LIN {X 0,Y 417.431,Z 307.432,A -85,B 0,C 180,E1 -10178.471,E2 -10178.471} C_VEL
LIN {X 0,Y 417.765,Z 300.419,A -85,B 0,C 180,E1 -10179.929,E2 -10179.929} C_VEL
LIN {X 0,Y 418.265,Z 291.62,A -85,B 0,C 180,E1 -10181.387,E2 -10181.387} C_VEL
LIN {X 0,Y 418.822,Z 282.602,A -85,B 0,C 180,E1 -10182.6,E2 -10182.6} C_VEL
LIN {X 0,Y 419.415,Z 273.392,A -85,B 0,C 180,E1 -10183.617,E2 -10183.617} C_VEL
LIN {X 0,Y 420.017,Z 263.241,A -85,B 0,C 180,E1 -10184.536,E2 -10184.536} C_VEL
LIN {X 0,Y 420.775,Z 251.442,A -85,B 0,C 180,E1 -10185.376,E2 -10185.376} C_VEL
LIN {X 0,Y 421.386,Z 239.15,A -85,B 0,C 180,E1 -10186.035,E2 -10186.035} C_VEL
LIN {X 0,Y 421.966,Z 225.694,A -85,B 0,C 180,E1 -10186.541,E2 -10186.541} C_VEL
LIN {X 0,Y 422.2,Z 212.111,A -85,B 0,C 180,E1 -10186.843,E2 -10186.843} C_VEL
LIN {X 0,Y 422.884,Z 138.438,A -85,B 0,C 180,E1 -10188.089,E2 -10188.089} C_VEL
LIN {X 0,Y 419.21,Z 111.774,A -85,B 0,C 180,E1 -10188.701,E2 -10188.701} C_VEL
LIN {X 0,Y 420.191,Z 93.552,A -85,B 0,C 180,E1 -10192.106,E2 -10192.106} C_VEL
LIN {X 0,Y 421.025,Z 79.98,A -85,B 0,C 180,E1 -10194.665,E2 -10194.665} C_VEL
LIN {X 0,Y 418.784,Z 67.568,A -85,B 0,C 180,E1 -10197.197,E2 -10197.197} C_VEL
LIN {X 0,Y 418.347,Z 65.37,A -85,B 0,C 180,E1 -10197.691,E2 -10197.691} C_VEL
LIN {X 0,Y 418.212,Z 65.388,A -85,B 0,C 180,E1 -10201.396,E2 -10201.396} C_VEL
LIN {X 0,Y 418.266,Z 65.381,A -85,B 0,C 180,E1 -10204.58,E2 -10204.58} C_VEL
LIN {X 0,Y 418.235,Z 65.39,A -85,B 0,C 180,E1 -10207.834,E2 -10207.834} C_VEL
LIN {X 0,Y 418.223,Z 65.386,A -85,B 0,C 180,E1 -10210.948,E2 -10210.948} C_VEL
LIN {X 0,Y 418.21,Z 65.392,A -85,B 0,C 180,E1 -10213.729,E2 -10213.729} C_VEL
LIN {X 0,Y 418.208,Z 65.387,A -85,B 0,C 180,E1 -10216.448,E2 -10216.448} C_VEL
LIN {X 0,Y 418.222,Z 65.39,A -85,B 0,C 180,E1 -10219.13,E2 -10219.13} C_VEL
LIN {X 0,Y 418.226,Z 65.385,A -85,B 0,C 180,E1 -10222.167,E2 -10222.167} C_VEL
LIN {X 0,Y 418.265,Z 65.385,A -85,B 0,C 180,E1 -10225.42,E2 -10225.42} C_VEL
LIN {X 0,Y 418.211,Z 65.389,A -85,B 0,C 180,E1 -10228.604,E2 -10228.604} C_VEL
LIN {X 0,Y 418.291,Z 65.377,A -85,B 0,C 180,E1 -10231.937,E2 -10231.937} C_VEL
LIN {X 0,Y 418.289,Z 65.381,A -85,B 0,C 180,E1 -10235.163,E2 -10235.163} C_VEL
LIN {X 0,Y 418.233,Z 65.386,A -85,B 0,C 180,E1 -10238.304,E2 -10238.304} C_VEL
LIN {X 0,Y 418.275,Z 65.38,A -85,B 0,C 180,E1 -10241.383,E2 -10241.383} C_VEL
LIN {X 0,Y 418.301,Z 65.381,A -85,B 0,C 180,E1 -10244.406,E2 -10244.406} C_VEL
LIN {X 0,Y 418.355,Z 65.369,A -85,B 0,C 180,E1 -10247.386,E2 -10247.386} C_VEL
LIN {X 0,Y 418.399,Z 65.363,A -85,B 0,C 180,E1 -10251.305,E2 -10251.305} C_VEL
LIN {X 0,Y 418.509,Z 65.356,A -85,B 0,C 180,E1 -10254.217,E2 -10254.217} C_VEL
LIN {X 0,Y 418.539,Z 65.352,A -85,B 0,C 180,E1 -10258.076,E2 -10258.076} C_VEL
LIN {X 0,Y 418.668,Z 65.336,A -85,B 0,C 180,E1 -10260,E2 -10260} C_VEL
LIN {X 0,Y 418.494,Z 65.352,A -85,B 0,C 180,E1 -10262.888,E2 -10262.888} C_VEL
LIN {X 0,Y 418.457,Z 65.356,A -85,B 0,C 180,E1 -10266.516,E2 -10266.516} C_VEL
LIN {X 0,Y 418.338,Z 65.377,A -85,B 0,C 180,E1 -10269.672,E2 -10269.672} C_VEL
LIN {X 0,Y 418.346,Z 65.371,A -85,B 0,C 180,E1 -10273.001,E2 -10273.001} C_VEL
LIN {X 0,Y 418.312,Z 65.374,A -85,B 0,C 180,E1 -10276.735,E2 -10276.735} C_VEL
LIN {X 0,Y 418.27,Z 65.383,A -85,B 0,C 180,E1 -10279.79,E2 -10279.79} C_VEL
LIN {X 0,Y 418.237,Z 65.385,A -85,B 0,C 180,E1 -10282.737,E2 -10282.737} C_VEL
LIN {X 0,Y 418.261,Z 65.382,A -85,B 0,C 180,E1 -10285.905,E2 -10285.905} C_VEL
LIN {X 0,Y 418.269,Z 65.386,A -85,B 0,C 180,E1 -10289.105,E2 -10289.105} C_VEL
LIN {X 0,Y 418.258,Z 65.386,A -85,B 0,C 180,E1 -10292.844,E2 -10292.844} C_VEL
LIN {X 0,Y 418.245,Z 65.383,A -85,B 0,C 180,E1 -10296.238,E2 -10296.238} C_VEL
LIN {X 0,Y 418.21,Z 65.387,A -85,B 0,C 180,E1 -10299.687,E2 -10299.687} C_VEL
LIN {X 0,Y 418.213,Z 65.389,A -85,B 0,C 180,E1 -10302.319,E2 -10302.319} C_VEL
LIN {X 0,Y 418.237,Z 65.386,A -85,B 0,C 180,E1 -10305.109,E2 -10305.109} C_VEL
LIN {X 0,Y 418.236,Z 65.384,A -85,B 0,C 180,E1 -10307.767,E2 -10307.767} C_VEL
LIN {X 0,Y 418.24,Z 65.383,A -85,B 0,C 180,E1 -10311.557,E2 -10311.557} C_VEL
LIN {X 0,Y 418.261,Z 65.381,A -85,B 0,C 180,E1 -10315.159,E2 -10315.159} C_VEL
LIN {X 0,Y 418.248,Z 65.383,A -85,B 0,C 180,E1 -10317.472,E2 -10317.472} C_VEL
LIN {X 0,Y 418.267,Z 65.38,A -85,B 0,C 180,E1 -10320.897,E2 -10320.897} C_VEL
LIN {X 0,Y 418.234,Z 65.391,A -85,B 0,C 180,E1 -10324.094,E2 -10324.094} C_VEL
LIN {X 0,Y 418.233,Z 65.385,A -85,B 0,C 180,E1 -10327.264,E2 -10327.264} C_VEL
LIN {X 0,Y 418.287,Z 65.379,A -85,B 0,C 180,E1 -10330.365,E2 -10330.365} C_VEL
LIN {X 0,Y 418.32,Z 65.376,A -85,B 0,C 180,E1 -10333.405,E2 -10333.405} C_VEL
LIN {X 0,Y 418.343,Z 65.434,A -85,B 0,C 180,E1 -10335.653,E2 -10335.653} C_VEL
LIN {X 0,Y 419.814,Z 74.736,A -85,B 0,C 180,E1 -10337.921,E2 -10337.921} C_VEL
LIN {X 0,Y 419.849,Z 76.846,A -85,B 0,C 180,E1 -10338.412,E2 -10338.412} C_VEL
LIN {X 0,Y 423.359,Z 95.58,A -85,B 0,C 180,E1 -10338.881,E2 -10338.881} C_VEL
LIN {X 0,Y 422.292,Z 183.825,A -85,B 0,C 180,E1 -10340.392,E2 -10340.392} C_VEL
LIN {X 0,Y 422.034,Z 197.591,A -85,B 0,C 180,E1 -10340.837,E2 -10340.837} C_VEL
LIN {X 0,Y 421.56,Z 210.007,A -85,B 0,C 180,E1 -10341.431,E2 -10341.431} C_VEL
LIN {X 0,Y 421.142,Z 221.833,A -85,B 0,C 180,E1 -10342.208,E2 -10342.208} C_VEL
LIN {X 0,Y 420.759,Z 228.414,A -85,B 0,C 180,E1 -10342.732,E2 -10342.732} C_VEL
LIN {X 0,Y 419.76,Z 233.376,A -85,B 0,C 180,E1 -10343.151,E2 -10343.151} C_VEL
LIN {X 0,Y 416.395,Z 241.174,A -85,B 0,C 180,E1 -10343.859,E2 -10343.859} C_VEL
LIN {X 0,Y 413.103,Z 248.473,A -85,B 0,C 180,E1 -10344.664,E2 -10344.664} C_VEL
LIN {X 0,Y 412.224,Z 252.648,A -85,B 0,C 180,E1 -10345.229,E2 -10345.229} C_VEL
LIN {X 0,Y 411.575,Z 261.003,A -85,B 0,C 180,E1 -10346.574,E2 -10346.574} C_VEL
LIN {X 0,Y 411.024,Z 268.36,A -85,B 0,C 180,E1 -10348.041,E2 -10348.041} C_VEL
LIN {X 0,Y 410.67,Z 274.265,A -85,B 0,C 180,E1 -10349.51,E2 -10349.51} C_VEL
LIN {X 0,Y 410.324,Z 278.946,A -85,B 0,C 180,E1 -10350.982,E2 -10350.982} C_VEL
LIN {X 0,Y 410.218,Z 282.523,A -85,B 0,C 180,E1 -10352.455,E2 -10352.455} C_VEL
LIN {X 0,Y 410.051,Z 285.111,A -85,B 0,C 180,E1 -10353.931,E2 -10353.931} C_VEL
LIN {X 0,Y 410.061,Z 286.328,A -85,B 0,C 180,E1 -10354.916,E2 -10354.916} C_VEL
LIN {X 0,Y 410.118,Z 287.328,A -85,B 0,C 180,E1 -10356.318,E2 -10356.318} C_VEL
LIN {X 0,Y 409.997,Z 287.526,A -85,B 0,C 180,E1 -10357.882,E2 -10357.882} C_VEL
LIN {X 0,Y 410.023,Z 287.151,A -85,B 0,C 180,E1 -10358.874,E2 -10358.874} C_VEL
LIN {X 0,Y 410.015,Z 286.357,A -85,B 0,C 180,E1 -10359.87,E2 -10359.87} C_VEL
LIN {X 0,Y 410.13,Z 285.135,A -85,B 0,C 180,E1 -10360.865,E2 -10360.865} C_VEL
LIN {X 0,Y 410.448,Z 282.065,A -85,B 0,C 180,E1 -10362.576,E2 -10362.576} C_VEL
LIN {X 0,Y 410.797,Z 277.448,A -85,B 0,C 180,E1 -10364.364,E2 -10364.364} C_VEL
LIN {X 0,Y 411.381,Z 271.232,A -85,B 0,C 180,E1 -10366.118,E2 -10366.118} C_VEL
LIN {X 0,Y 411.974,Z 264.461,A -85,B 0,C 180,E1 -10367.619,E2 -10367.619} C_VEL
LIN {X 0,Y 412.633,Z 257.443,A -85,B 0,C 180,E1 -10368.882,E2 -10368.882} C_VEL
LIN {X 0,Y 413.43,Z 248.997,A -85,B 0,C 180,E1 -10370.135,E2 -10370.135} C_VEL
LIN {X 0,Y 414.152,Z 239.692,A -85,B 0,C 180,E1 -10371.268,E2 -10371.268} C_VEL
LIN {X 0,Y 414.956,Z 229.493,A -85,B 0,C 180,E1 -10372.27,E2 -10372.27} C_VEL
LIN {X 0,Y 415.733,Z 218.335,A -85,B 0,C 180,E1 -10373.144,E2 -10373.144} C_VEL
LIN {X 0,Y 416.464,Z 205.903,A -85,B 0,C 180,E1 -10373.892,E2 -10373.892} C_VEL
LIN {X 0,Y 416.995,Z 192.882,A -85,B 0,C 180,E1 -10374.445,E2 -10374.445} C_VEL
LIN {X 0,Y 417.333,Z 179.624,A -85,B 0,C 180,E1 -10374.8,E2 -10374.8} C_VEL
LIN {X 0,Y 418.439,Z 96.881,A -85,B 0,C 180,E1 -10376.241,E2 -10376.241} C_VEL
LIN {X 0,Y 414.203,Z 79.905,A -85,B 0,C 180,E1 -10376.788,E2 -10376.788} C_VEL
LIN {X 0,Y 413.433,Z 77.348,A -85,B 0,C 180,E1 -10376.906,E2 -10376.906} C_VEL
LIN {X 0,Y 411.219,Z 66.264,A -85,B 0,C 180,E1 -10379.817,E2 -10379.817} C_VEL
LIN {X 0,Y 411.206,Z 66.265,A -85,B 0,C 180,E1 -10383.156,E2 -10383.156} C_VEL
LIN {X 0,Y 411.191,Z 66.265,A -85,B 0,C 180,E1 -10386.551,E2 -10386.551} C_VEL
LIN {X 0,Y 411.17,Z 66.27,A -85,B 0,C 180,E1 -10389.72,E2 -10389.72} C_VEL
LIN {X 0,Y 411.164,Z 66.268,A -85,B 0,C 180,E1 -10393.135,E2 -10393.135} C_VEL
LIN {X 0,Y 411.166,Z 66.264,A -85,B 0,C 180,E1 -10395.882,E2 -10395.882} C_VEL
LIN {X 0,Y 411.149,Z 66.265,A -85,B 0,C 180,E1 -10398.775,E2 -10398.775} C_VEL
LIN {X 0,Y 411.179,Z 66.266,A -85,B 0,C 180,E1 -10402.024,E2 -10402.024} C_VEL
LIN {X 0,Y 411.202,Z 66.261,A -85,B 0,C 180,E1 -10405.124,E2 -10405.124} C_VEL
LIN {X 0,Y 411.156,Z 66.263,A -85,B 0,C 180,E1 -10408.001,E2 -10408.001} C_VEL
LIN {X 0,Y 411.17,Z 66.266,A -85,B 0,C 180,E1 -10411.406,E2 -10411.406} C_VEL
LIN {X 0,Y 411.19,Z 66.267,A -85,B 0,C 180,E1 -10414.941,E2 -10414.941} C_VEL
LIN {X 0,Y 411.206,Z 66.256,A -85,B 0,C 180,E1 -10417.913,E2 -10417.913} C_VEL
LIN {X 0,Y 411.222,Z 66.258,A -85,B 0,C 180,E1 -10421.051,E2 -10421.051} C_VEL
LIN {X 0,Y 411.25,Z 66.254,A -85,B 0,C 180,E1 -10424.131,E2 -10424.131} C_VEL
LIN {X 0,Y 411.307,Z 66.242,A -85,B 0,C 180,E1 -10427.165,E2 -10427.165} C_VEL
LIN {X 0,Y 411.29,Z 66.251,A -85,B 0,C 180,E1 -10430.161,E2 -10430.161} C_VEL
LIN {X 0,Y 411.389,Z 66.231,A -85,B 0,C 180,E1 -10433.132,E2 -10433.132} C_VEL
LIN {X 0,Y 411.291,Z 66.248,A -85,B 0,C 180,E1 -10435.099,E2 -10435.099} C_VEL
LIN {X 0,Y 411.509,Z 66.227,A -85,B 0,C 180,E1 -10438.042,E2 -10438.042} C_VEL
LIN {X 0,Y 411.439,Z 66.228,A -85,B 0,C 180,E1 -10440.979,E2 -10440.979} C_VEL
LIN {X 0,Y 411.432,Z 66.233,A -85,B 0,C 180,E1 -10442.937,E2 -10442.937} C_VEL
LIN {X 0,Y 411.432,Z 66.227,A -85,B 0,C 180,E1 -10445.882,E2 -10445.882} C_VEL
LIN {X 0,Y 411.32,Z 66.246,A -85,B 0,C 180,E1 -10448.846,E2 -10448.846} C_VEL
LIN {X 0,Y 411.286,Z 66.246,A -85,B 0,C 180,E1 -10451.833,E2 -10451.833} C_VEL
LIN {X 0,Y 411.258,Z 66.253,A -85,B 0,C 180,E1 -10454.853,E2 -10454.853} C_VEL
LIN {X 0,Y 411.246,Z 66.255,A -85,B 0,C 180,E1 -10457.915,E2 -10457.915} C_VEL
LIN {X 0,Y 411.199,Z 66.263,A -85,B 0,C 180,E1 -10461.034,E2 -10461.034} C_VEL
LIN {X 0,Y 411.22,Z 66.259,A -85,B 0,C 180,E1 -10464.216,E2 -10464.216} C_VEL
LIN {X 0,Y 411.261,Z 66.255,A -85,B 0,C 180,E1 -10467.477,E2 -10467.477} C_VEL
LIN {X 0,Y 411.192,Z 66.263,A -85,B 0,C 180,E1 -10470.847,E2 -10470.847} C_VEL
LIN {X 0,Y 411.209,Z 66.26,A -85,B 0,C 180,E1 -10474.333,E2 -10474.333} C_VEL
LIN {X 0,Y 411.195,Z 66.256,A -85,B 0,C 180,E1 -10477.974,E2 -10477.974} C_VEL
LIN {X 0,Y 411.166,Z 66.267,A -85,B 0,C 180,E1 -10481.228,E2 -10481.228} C_VEL
LIN {X 0,Y 411.178,Z 66.268,A -85,B 0,C 180,E1 -10484.49,E2 -10484.49} C_VEL
LIN {X 0,Y 411.18,Z 66.265,A -85,B 0,C 180,E1 -10488.194,E2 -10488.194} C_VEL
LIN {X 0,Y 411.225,Z 66.26,A -85,B 0,C 180,E1 -10490.776,E2 -10490.776} C_VEL
LIN {X 0,Y 411.2,Z 66.259,A -85,B 0,C 180,E1 -10494.471,E2 -10494.471} C_VEL
LIN {X 0,Y 411.21,Z 66.267,A -85,B 0,C 180,E1 -10496.873,E2 -10496.873} C_VEL
LIN {X 0,Y 411.235,Z 66.265,A -85,B 0,C 180,E1 -10500.644,E2 -10500.644} C_VEL
LIN {X 0,Y 411.251,Z 66.323,A -85,B 0,C 180,E1 -10500.882,E2 -10500.882} C_VEL
LIN {X 0,Y 413.861,Z 78.061,A -85,B 0,C 180,E1 -10503.527,E2 -10503.527} C_VEL
LIN {X 0,Y 415.004,Z 84.662,A -85,B 0,C 180,E1 -10504.952,E2 -10504.952} C_VEL
LIN {X 0,Y 413.661,Z 101.777,A -85,B 0,C 180,E1 -10508.313,E2 -10508.313} C_VEL
LIN {X 0,Y 413.058,Z 111.347,A -85,B 0,C 180,E1 -10510.146,E2 -10510.146} C_VEL
LIN {X 0,Y 417.432,Z 136.961,A -85,B 0,C 180,E1 -10510.852,E2 -10510.852} C_VEL
LIN {X 0,Y 417.89,Z 142.841,A -85,B 0,C 180,E1 -10510.983,E2 -10510.983} C_VEL
LIN {X 0,Y 416.919,Z 219.576,A -85,B 0,C 180,E1 -10512.336,E2 -10512.336} C_VEL
LIN {X 0,Y 416.286,Z 232.903,A -85,B 0,C 180,E1 -10512.752,E2 -10512.752} C_VEL
LIN {X 0,Y 415.492,Z 245.646,A -85,B 0,C 180,E1 -10513.351,E2 -10513.351} C_VEL
LIN {X 0,Y 414.638,Z 257.78,A -85,B 0,C 180,E1 -10514.138,E2 -10514.138} C_VEL
LIN {X 0,Y 413.688,Z 269.312,A -85,B 0,C 180,E1 -10515.11,E2 -10515.11} C_VEL
LIN {X 0,Y 412.753,Z 279.713,A -85,B 0,C 180,E1 -10516.209,E2 -10516.209} C_VEL
LIN {X 0,Y 412.052,Z 289.098,A -85,B 0,C 180,E1 -10517.439,E2 -10517.439} C_VEL
LIN {X 0,Y 411.212,Z 298.174,A -85,B 0,C 180,E1 -10518.914,E2 -10518.914} C_VEL
LIN {X 0,Y 410.659,Z 305.511,A -85,B 0,C 180,E1 -10520.394,E2 -10520.394} C_VEL
LIN {X 0,Y 410.257,Z 312.261,A -85,B 0,C 180,E1 -10522.123,E2 -10522.123} C_VEL
LIN {X 0,Y 410.047,Z 317.157,A -85,B 0,C 180,E1 -10523.77,E2 -10523.77} C_VEL
LIN {X 0,Y 410.002,Z 320.138,A -85,B 0,C 180,E1 -10525.083,E2 -10525.083} C_VEL
LIN {X 0,Y 409.97,Z 323.132,A -85,B 0,C 180,E1 -10527.052,E2 -10527.052} C_VEL
LIN {X 0,Y 410.02,Z 324.037,A -85,B 0,C 180,E1 -10528.035,E2 -10528.035} C_VEL
LIN {X 0,Y 409.984,Z 324.507,A -85,B 0,C 180,E1 -10529.017,E2 -10529.017} C_VEL
LIN {X 0,Y 409.981,Z 324.574,A -85,B 0,C 180,E1 -10530,E2 -10530} C_VEL
LIN {X 0,Y 410.024,Z 323.546,A -85,B 0,C 180,E1 -10531.964,E2 -10531.964} C_VEL
LIN {X 0,Y 410.012,Z 322.408,A -85,B 0,C 180,E1 -10532.947,E2 -10532.947} C_VEL
LIN {X 0,Y 409.959,Z 320.83,A -85,B 0,C 180,E1 -10533.932,E2 -10533.932} C_VEL
LIN {X 0,Y 410,Z 317.661,A -85,B 0,C 180,E1 -10535.409,E2 -10535.409} C_VEL
LIN {X 0,Y 410.076,Z 313.415,A -85,B 0,C 180,E1 -10536.89,E2 -10536.89} C_VEL
LIN {X 0,Y 410.353,Z 306.957,A -85,B 0,C 180,E1 -10538.618,E2 -10538.618} C_VEL
LIN {X 0,Y 410.702,Z 299.897,A -85,B 0,C 180,E1 -10540.102,E2 -10540.102} C_VEL
LIN {X 0,Y 411.266,Z 291.048,A -85,B 0,C 180,E1 -10541.583,E2 -10541.583} C_VEL
LIN {X 0,Y 411.876,Z 281.981,A -85,B 0,C 180,E1 -10542.816,E2 -10542.816} C_VEL
LIN {X 0,Y 412.549,Z 272.003,A -85,B 0,C 180,E1 -10543.923,E2 -10543.923} C_VEL
LIN {X 0,Y 413.228,Z 260.922,A -85,B 0,C 180,E1 -10544.906,E2 -10544.906} C_VEL
LIN {X 0,Y 413.978,Z 248.494,A -85,B 0,C 180,E1 -10545.761,E2 -10545.761} C_VEL
LIN {X 0,Y 414.567,Z 236.704,A -85,B 0,C 180,E1 -10546.37,E2 -10546.37} C_VEL
LIN {X 0,Y 415.167,Z 224.022,A -85,B 0,C 180,E1 -10546.82,E2 -10546.82} C_VEL
LIN {X 0,Y 415.431,Z 207.762,A -85,B 0,C 180,E1 -10547.157,E2 -10547.157} C_VEL
LIN {X 0,Y 415.989,Z 138.503,A -85,B 0,C 180,E1 -10548.353,E2 -10548.353} C_VEL
LIN {X 0,Y 412.261,Z 111.404,A -85,B 0,C 180,E1 -10548.996,E2 -10548.996} C_VEL
LIN {X 0,Y 413.316,Z 93.017,A -85,B 0,C 180,E1 -10552.494,E2 -10552.494} C_VEL
LIN {X 0,Y 414.043,Z 80.793,A -85,B 0,C 180,E1 -10554.841,E2 -10554.841} C_VEL
LIN {X 0,Y 411.705,Z 68.288,A -85,B 0,C 180,E1 -10557.445,E2 -10557.445} C_VEL
LIN {X 0,Y 411.306,Z 66.246,A -85,B 0,C 180,E1 -10557.889,E2 -10557.889} C_VEL
LIN {X 0,Y 411.183,Z 66.263,A -85,B 0,C 180,E1 -10561.283,E2 -10561.283} C_VEL
LIN {X 0,Y 411.206,Z 66.261,A -85,B 0,C 180,E1 -10564.333,E2 -10564.333} C_VEL
LIN {X 0,Y 411.201,Z 66.264,A -85,B 0,C 180,E1 -10567.973,E2 -10567.973} C_VEL
LIN {X 0,Y 411.183,Z 66.263,A -85,B 0,C 180,E1 -10570.504,E2 -10570.504} C_VEL
LIN {X 0,Y 411.173,Z 66.266,A -85,B 0,C 180,E1 -10573.133,E2 -10573.133} C_VEL
LIN {X 0,Y 411.167,Z 66.267,A -85,B 0,C 180,E1 -10575.881,E2 -10575.881} C_VEL
LIN {X 0,Y 411.162,Z 66.266,A -85,B 0,C 180,E1 -10578.772,E2 -10578.772} C_VEL
LIN {X 0,Y 411.192,Z 66.262,A -85,B 0,C 180,E1 -10582.026,E2 -10582.026} C_VEL
LIN {X 0,Y 411.205,Z 66.262,A -85,B 0,C 180,E1 -10585.666,E2 -10585.666} C_VEL
LIN {X 0,Y 411.189,Z 66.268,A -85,B 0,C 180,E1 -10589.152,E2 -10589.152} C_VEL
LIN {X 0,Y 411.258,Z 66.255,A -85,B 0,C 180,E1 -10592.522,E2 -10592.522} C_VEL
LIN {X 0,Y 411.226,Z 66.257,A -85,B 0,C 180,E1 -10595.785,E2 -10595.785} C_VEL
LIN {X 0,Y 411.196,Z 66.265,A -85,B 0,C 180,E1 -10598.966,E2 -10598.966} C_VEL
LIN {X 0,Y 411.245,Z 66.256,A -85,B 0,C 180,E1 -10602.085,E2 -10602.085} C_VEL
LIN {X 0,Y 411.259,Z 66.254,A -85,B 0,C 180,E1 -10605.147,E2 -10605.147} C_VEL
LIN {X 0,Y 411.283,Z 66.254,A -85,B 0,C 180,E1 -10608.167,E2 -10608.167} C_VEL
LIN {X 0,Y 411.44,Z 66.236,A -85,B 0,C 180,E1 -10612.189,E2 -10612.189} C_VEL
LIN {X 0,Y 411.471,Z 66.232,A -85,B 0,C 180,E1 -10614.118,E2 -10614.118} C_VEL
LIN {X 0,Y 411.508,Z 66.228,A -85,B 0,C 180,E1 -10618.043,E2 -10618.043} C_VEL
LIN {X 0,Y 411.638,Z 66.212,A -85,B 0,C 180,E1 -10620,E2 -10620} C_VEL
LIN {X 0,Y 411.451,Z 66.229,A -85,B 0,C 180,E1 -10622.938,E2 -10622.938} C_VEL
LIN {X 0,Y 411.422,Z 66.233,A -85,B 0,C 180,E1 -10626.514,E2 -10626.514} C_VEL
LIN {X 0,Y 411.291,Z 66.255,A -85,B 0,C 180,E1 -10629.839,E2 -10629.839} C_VEL
LIN {X 0,Y 411.305,Z 66.248,A -85,B 0,C 180,E1 -10633.104,E2 -10633.104} C_VEL
LIN {X 0,Y 411.257,Z 66.254,A -85,B 0,C 180,E1 -10636.889,E2 -10636.889} C_VEL
LIN {X 0,Y 411.231,Z 66.258,A -85,B 0,C 180,E1 -10639.987,E2 -10639.987} C_VEL
LIN {X 0,Y 411.202,Z 66.265,A -85,B 0,C 180,E1 -10643.148,E2 -10643.148} C_VEL
LIN {X 0,Y 411.234,Z 66.256,A -85,B 0,C 180,E1 -10646.382,E2 -10646.382} C_VEL
LIN {X 0,Y 411.201,Z 66.262,A -85,B 0,C 180,E1 -10649.713,E2 -10649.713} C_VEL
LIN {X 0,Y 411.207,Z 66.265,A -85,B 0,C 180,E1 -10653.156,E2 -10653.156} C_VEL
LIN {X 0,Y 411.193,Z 66.264,A -85,B 0,C 180,E1 -10656.553,E2 -10656.553} C_VEL
LIN {X 0,Y 411.178,Z 66.263,A -85,B 0,C 180,E1 -10659.722,E2 -10659.722} C_VEL
LIN {X 0,Y 411.165,Z 66.267,A -85,B 0,C 180,E1 -10663.135,E2 -10663.135} C_VEL
LIN {X 0,Y 411.169,Z 66.265,A -85,B 0,C 180,E1 -10665.882,E2 -10665.882} C_VEL
LIN {X 0,Y 411.16,Z 66.27,A -85,B 0,C 180,E1 -10668.773,E2 -10668.773} C_VEL
LIN {X 0,Y 411.188,Z 66.264,A -85,B 0,C 180,E1 -10672.026,E2 -10672.026} C_VEL
LIN {X 0,Y 411.208,Z 66.26,A -85,B 0,C 180,E1 -10675.667,E2 -10675.667} C_VEL
LIN {X 0,Y 411.191,Z 66.261,A -85,B 0,C 180,E1 -10679.153,E2 -10679.153} C_VEL
LIN {X 0,Y 411.191,Z 66.264,A -85,B 0,C 180,E1 -10682.518,E2 -10682.518} C_VEL
LIN {X 0,Y 411.199,Z 66.265,A -85,B 0,C 180,E1 -10685.783,E2 -10685.783} C_VEL
LIN {X 0,Y 411.2,Z 66.26,A -85,B 0,C 180,E1 -10688.966,E2 -10688.966} C_VEL
LIN {X 0,Y 411.253,Z 66.261,A -85,B 0,C 180,E1 -10692.085,E2 -10692.085} C_VEL
LIN {X 0,Y 411.297,Z 66.336,A -85,B 0,C 180,E1 -10695.465,E2 -10695.465} C_VEL
LIN {X 0,Y 412.794,Z 75.399,A -85,B 0,C 180,E1 -10697.713,E2 -10697.713} C_VEL
LIN {X 0,Y 412.884,Z 77.112,A -85,B 0,C 180,E1 -10698.121,E2 -10698.121} C_VEL
LIN {X 0,Y 416.531,Z 96.247,A -85,B 0,C 180,E1 -10698.619,E2 -10698.619} C_VEL
LIN {X 0,Y 415.451,Z 183.74,A -85,B 0,C 180,E1 -10700.138,E2 -10700.138} C_VEL
LIN {X 0,Y 415.189,Z 196.938,A -85,B 0,C 180,E1 -10700.562,E2 -10700.562} C_VEL
LIN {X 0,Y 414.713,Z 209.605,A -85,B 0,C 180,E1 -10701.166,E2 -10701.166} C_VEL
LIN {X 0,Y 414.258,Z 221.649,A -85,B 0,C 180,E1 -10701.955,E2 -10701.955} C_VEL
LIN {X 0,Y 413.527,Z 233.103,A -85,B 0,C 180,E1 -10702.923,E2 -10702.923} C_VEL
LIN {X 0,Y 412.847,Z 243.412,A -85,B 0,C 180,E1 -10704.015,E2 -10704.015} C_VEL
LIN {X 0,Y 412.224,Z 252.648,A -85,B 0,C 180,E1 -10705.229,E2 -10705.229} C_VEL
LIN {X 0,Y 411.354,Z 256.67,A -85,B 0,C 180,E1 -10705.822,E2 -10705.822} C_VEL
LIN {X 0,Y 408.095,Z 262.811,A -85,B 0,C 180,E1 -10706.806,E2 -10706.806} C_VEL
LIN {X 0,Y 404.771,Z 268.376,A -85,B 0,C 180,E1 -10707.869,E2 -10707.869} C_VEL
LIN {X 0,Y 403.817,Z 271.416,A -85,B 0,C 180,E1 -10708.576,E2 -10708.576} C_VEL
LIN {X 0,Y 403.389,Z 276.545,A -85,B 0,C 180,E1 -10710,E2 -10710} C_VEL
LIN {X 0,Y 403.227,Z 280.774,A -85,B 0,C 180,E1 -10711.498,E2 -10711.498} C_VEL
LIN {X 0,Y 403.107,Z 283.96,A -85,B 0,C 180,E1 -10712.998,E2 -10712.998} C_VEL
LIN {X 0,Y 402.961,Z 285.554,A -85,B 0,C 180,E1 -10714.001,E2 -10714.001} C_VEL
LIN {X 0,Y 402.992,Z 286.738,A -85,B 0,C 180,E1 -10715.003,E2 -10715.003} C_VEL
LIN {X 0,Y 403.02,Z 287.619,A -85,B 0,C 180,E1 -10716.282,E2 -10716.282} C_VEL
LIN {X 0,Y 402.924,Z 287.834,A -85,B 0,C 180,E1 -10718.022,E2 -10718.022} C_VEL
LIN {X 0,Y 402.926,Z 287.428,A -85,B 0,C 180,E1 -10719.032,E2 -10719.032} C_VEL
LIN {X 0,Y 402.939,Z 286.584,A -85,B 0,C 180,E1 -10720.045,E2 -10720.045} C_VEL
LIN {X 0,Y 403.082,Z 285.334,A -85,B 0,C 180,E1 -10721.058,E2 -10721.058} C_VEL
LIN {X 0,Y 403.395,Z 282.477,A -85,B 0,C 180,E1 -10722.67,E2 -10722.67} C_VEL
LIN {X 0,Y 403.659,Z 278.966,A -85,B 0,C 180,E1 -10724.108,E2 -10724.108} C_VEL
LIN {X 0,Y 404.162,Z 274.114,A -85,B 0,C 180,E1 -10725.637,E2 -10725.637} C_VEL
LIN {X 0,Y 404.821,Z 267.456,A -85,B 0,C 180,E1 -10727.283,E2 -10727.283} C_VEL
LIN {X 0,Y 405.462,Z 260.258,A -85,B 0,C 180,E1 -10728.704,E2 -10728.704} C_VEL
LIN {X 0,Y 406.287,Z 252.316,A -85,B 0,C 180,E1 -10729.977,E2 -10729.977} C_VEL
LIN {X 0,Y 407.15,Z 242.571,A -85,B 0,C 180,E1 -10731.254,E2 -10731.254} C_VEL
LIN {X 0,Y 408.047,Z 231.69,A -85,B 0,C 180,E1 -10732.4,E2 -10732.4} C_VEL
LIN {X 0,Y 408.862,Z 221.048,A -85,B 0,C 180,E1 -10733.288,E2 -10733.288} C_VEL
LIN {X 0,Y 409.615,Z 209.292,A -85,B 0,C 180,E1 -10734.048,E2 -10734.048} C_VEL
LIN {X 0,Y 410.214,Z 196.342,A -85,B 0,C 180,E1 -10734.664,E2 -10734.664} C_VEL
LIN {X 0,Y 410.64,Z 184.095,A -85,B 0,C 180,E1 -10735.049,E2 -10735.049} C_VEL
LIN {X 0,Y 411.784,Z 97.678,A -85,B 0,C 180,E1 -10736.598,E2 -10736.598} C_VEL
LIN {X 0,Y 407.848,Z 82.078,A -85,B 0,C 180,E1 -10737.116,E2 -10737.116} C_VEL
LIN {X 0,Y 406.304,Z 77.665,A -85,B 0,C 180,E1 -10737.321,E2 -10737.321} C_VEL
LIN {X 0,Y 404.176,Z 67.142,A -85,B 0,C 180,E1 -10740.146,E2 -10740.146} C_VEL
LIN {X 0,Y 404.139,Z 67.149,A -85,B 0,C 180,E1 -10743.813,E2 -10743.813} C_VEL
LIN {X 0,Y 404.133,Z 67.142,A -85,B 0,C 180,E1 -10746.874,E2 -10746.874} C_VEL
LIN {X 0,Y 404.121,Z 67.148,A -85,B 0,C 180,E1 -10750.075,E2 -10750.075} C_VEL
LIN {X 0,Y 404.144,Z 67.142,A -85,B 0,C 180,E1 -10753.082,E2 -10753.082} C_VEL
LIN {X 0,Y 404.123,Z 67.141,A -85,B 0,C 180,E1 -10755.922,E2 -10755.922} C_VEL
LIN {X 0,Y 404.103,Z 67.143,A -85,B 0,C 180,E1 -10758.632,E2 -10758.632} C_VEL
LIN {X 0,Y 404.136,Z 67.143,A -85,B 0,C 180,E1 -10761.496,E2 -10761.496} C_VEL
LIN {X 0,Y 404.173,Z 67.135,A -85,B 0,C 180,E1 -10764.982,E2 -10764.982} C_VEL
LIN {X 0,Y 404.133,Z 67.137,A -85,B 0,C 180,E1 -10768.444,E2 -10768.444} C_VEL
LIN {X 0,Y 404.15,Z 67.143,A -85,B 0,C 180,E1 -10770.862,E2 -10770.862} C_VEL
LIN {X 0,Y 404.154,Z 67.141,A -85,B 0,C 180,E1 -10774.723,E2 -10774.723} C_VEL
LIN {X 0,Y 404.169,Z 67.134,A -85,B 0,C 180,E1 -10777.508,E2 -10777.508} C_VEL
LIN {X 0,Y 404.165,Z 67.142,A -85,B 0,C 180,E1 -10780.707,E2 -10780.707} C_VEL
LIN {X 0,Y 404.22,Z 67.129,A -85,B 0,C 180,E1 -10783.848,E2 -10783.848} C_VEL
LIN {X 0,Y 404.287,Z 67.118,A -85,B 0,C 180,E1 -10786.939,E2 -10786.939} C_VEL
LIN {X 0,Y 404.256,Z 67.126,A -85,B 0,C 180,E1 -10789.988,E2 -10789.988} C_VEL
LIN {X 0,Y 404.34,Z 67.109,A -85,B 0,C 180,E1 -10793.011,E2 -10793.011} C_VEL
LIN {X 0,Y 404.262,Z 67.124,A -85,B 0,C 180,E1 -10795.013,E2 -10795.013} C_VEL
LIN {X 0,Y 404.478,Z 67.103,A -85,B 0,C 180,E1 -10798.008,E2 -10798.008} C_VEL
LIN {X 0,Y 404.404,Z 67.104,A -85,B 0,C 180,E1 -10800.996,E2 -10800.996} C_VEL
LIN {X 0,Y 404.392,Z 67.11,A -85,B 0,C 180,E1 -10802.988,E2 -10802.988} C_VEL
LIN {X 0,Y 404.38,Z 67.105,A -85,B 0,C 180,E1 -10805.985,E2 -10805.985} C_VEL
LIN {X 0,Y 404.267,Z 67.124,A -85,B 0,C 180,E1 -10809.001,E2 -10809.001} C_VEL
LIN {X 0,Y 404.259,Z 67.121,A -85,B 0,C 180,E1 -10812.041,E2 -10812.041} C_VEL
LIN {X 0,Y 404.205,Z 67.133,A -85,B 0,C 180,E1 -10815.118,E2 -10815.118} C_VEL
LIN {X 0,Y 404.206,Z 67.13,A -85,B 0,C 180,E1 -10818.238,E2 -10818.238} C_VEL
LIN {X 0,Y 404.141,Z 67.139,A -85,B 0,C 180,E1 -10821.419,E2 -10821.419} C_VEL
LIN {X 0,Y 404.175,Z 67.137,A -85,B 0,C 180,E1 -10824.666,E2 -10824.666} C_VEL
LIN {X 0,Y 404.197,Z 67.133,A -85,B 0,C 180,E1 -10827.999,E2 -10827.999} C_VEL
LIN {X 0,Y 404.142,Z 67.141,A -85,B 0,C 180,E1 -10831.558,E2 -10831.558} C_VEL
LIN {X 0,Y 404.187,Z 67.127,A -85,B 0,C 180,E1 -10835.016,E2 -10835.016} C_VEL
LIN {X 0,Y 404.155,Z 67.14,A -85,B 0,C 180,E1 -10838.757,E2 -10838.757} C_VEL
LIN {X 0,Y 404.125,Z 67.143,A -85,B 0,C 180,E1 -10841.599,E2 -10841.599} C_VEL
LIN {X 0,Y 404.147,Z 67.144,A -85,B 0,C 180,E1 -10844.522,E2 -10844.522} C_VEL
LIN {X 0,Y 404.139,Z 67.14,A -85,B 0,C 180,E1 -10847.295,E2 -10847.295} C_VEL
LIN {X 0,Y 404.171,Z 67.138,A -85,B 0,C 180,E1 -10849.955,E2 -10849.955} C_VEL
LIN {X 0,Y 404.139,Z 67.142,A -85,B 0,C 180,E1 -10853.125,E2 -10853.125} C_VEL
LIN {X 0,Y 404.147,Z 67.148,A -85,B 0,C 180,E1 -10856.188,E2 -10856.188} C_VEL
LIN {X 0,Y 404.148,Z 67.149,A -85,B 0,C 180,E1 -10859.715,E2 -10859.715} C_VEL
LIN {X 0,Y 404.184,Z 67.186,A -85,B 0,C 180,E1 -10860.524,E2 -10860.524} C_VEL
LIN {X 0,Y 406.654,Z 77.984,A -85,B 0,C 180,E1 -10863.02,E2 -10863.02} C_VEL
LIN {X 0,Y 408.092,Z 85.896,A -85,B 0,C 180,E1 -10864.771,E2 -10864.771} C_VEL
LIN {X 0,Y 406.83,Z 101.679,A -85,B 0,C 180,E1 -10867.93,E2 -10867.93} C_VEL
LIN {X 0,Y 406.177,Z 110.77,A -85,B 0,C 180,E1 -10869.731,E2 -10869.731} C_VEL
LIN {X 0,Y 410.77,Z 137.187,A -85,B 0,C 180,E1 -10870.496,E2 -10870.496} C_VEL
LIN {X 0,Y 411.275,Z 143.074,A -85,B 0,C 180,E1 -10870.632,E2 -10870.632} C_VEL
LIN {X 0,Y 410.225,Z 219.711,A -85,B 0,C 180,E1 -10872.009,E2 -10872.009} C_VEL
LIN {X 0,Y 409.589,Z 232.807,A -85,B 0,C 180,E1 -10872.429,E2 -10872.429} C_VEL
LIN {X 0,Y 408.712,Z 246.047,A -85,B 0,C 180,E1 -10873.067,E2 -10873.067} C_VEL
LIN {X 0,Y 407.82,Z 257.966,A -85,B 0,C 180,E1 -10873.866,E2 -10873.866} C_VEL
LIN {X 0,Y 406.82,Z 269.403,A -85,B 0,C 180,E1 -10874.853,E2 -10874.853} C_VEL
LIN {X 0,Y 405.854,Z 279.731,A -85,B 0,C 180,E1 -10875.97,E2 -10875.97} C_VEL
LIN {X 0,Y 405.106,Z 289.033,A -85,B 0,C 180,E1 -10877.221,E2 -10877.221} C_VEL
LIN {X 0,Y 404.198,Z 298.065,A -85,B 0,C 180,E1 -10878.719,E2 -10878.719} C_VEL
LIN {X 0,Y 403.621,Z 305.363,A -85,B 0,C 180,E1 -10880.225,E2 -10880.225} C_VEL
LIN {X 0,Y 403.191,Z 312.064,A -85,B 0,C 180,E1 -10881.984,E2 -10881.984} C_VEL
LIN {X 0,Y 402.94,Z 317.325,A -85,B 0,C 180,E1 -10883.818,E2 -10883.818} C_VEL
LIN {X 0,Y 402.91,Z 319.884,A -85,B 0,C 180,E1 -10884.996,E2 -10884.996} C_VEL
LIN {X 0,Y 402.868,Z 322.853,A -85,B 0,C 180,E1 -10887,E2 -10887} C_VEL
LIN {X 0,Y 402.948,Z 323.744,A -85,B 0,C 180,E1 -10888.001,E2 -10888.001} C_VEL
LIN {X 0,Y 402.908,Z 324.193,A -85,B 0,C 180,E1 -10889,E2 -10889} C_VEL
LIN {X 0,Y 402.903,Z 324.247,A -85,B 0,C 180,E1 -10890,E2 -10890} C_VEL
LIN {X 0,Y 402.953,Z 323.196,A -85,B 0,C 180,E1 -10891.999,E2 -10891.999} C_VEL
LIN {X 0,Y 402.911,Z 322.031,A -85,B 0,C 180,E1 -10892.999,E2 -10892.999} C_VEL
LIN {X 0,Y 402.913,Z 319.512,A -85,B 0,C 180,E1 -10894.502,E2 -10894.502} C_VEL
LIN {X 0,Y 402.885,Z 315.674,A -85,B 0,C 180,E1 -10896.109,E2 -10896.109} C_VEL
LIN {X 0,Y 403.093,Z 311.31,A -85,B 0,C 180,E1 -10897.513,E2 -10897.513} C_VEL
LIN {X 0,Y 403.394,Z 304.259,A -85,B 0,C 180,E1 -10899.274,E2 -10899.274} C_VEL
LIN {X 0,Y 403.815,Z 296.622,A -85,B 0,C 180,E1 -10900.783,E2 -10900.783} C_VEL
LIN {X 0,Y 404.421,Z 288.824,A -85,B 0,C 180,E1 -10902.036,E2 -10902.036} C_VEL
LIN {X 0,Y 405.041,Z 279.919,A -85,B 0,C 180,E1 -10903.216,E2 -10903.216} C_VEL
LIN {X 0,Y 405.704,Z 268.684,A -85,B 0,C 180,E1 -10904.419,E2 -10904.419} C_VEL
LIN {X 0,Y 406.564,Z 256.896,A -85,B 0,C 180,E1 -10905.413,E2 -10905.413} C_VEL
LIN {X 0,Y 407.312,Z 244.265,A -85,B 0,C 180,E1 -10906.219,E2 -10906.219} C_VEL
LIN {X 0,Y 407.941,Z 231.68,A -85,B 0,C 180,E1 -10906.804,E2 -10906.804} C_VEL
LIN {X 0,Y 408.408,Z 218.647,A -85,B 0,C 180,E1 -10907.203,E2 -10907.203} C_VEL
LIN {X 0,Y 409.186,Z 139.415,A -85,B 0,C 180,E1 -10908.605,E2 -10908.605} C_VEL
LIN {X 0,Y 405.301,Z 111.027,A -85,B 0,C 180,E1 -10909.302,E2 -10909.302} C_VEL
LIN {X 0,Y 406.534,Z 91.12,A -85,B 0,C 180,E1 -10913.159,E2 -10913.159} C_VEL
LIN {X 0,Y 407.099,Z 82.978,A -85,B 0,C 180,E1 -10914.749,E2 -10914.749} C_VEL
LIN {X 0,Y 405.26,Z 72.092,A -85,B 0,C 180,E1 -10917.037,E2 -10917.037} C_VEL
LIN {X 0,Y 404.257,Z 67.125,A -85,B 0,C 180,E1 -10918.136,E2 -10918.136} C_VEL
LIN {X 0,Y 404.14,Z 67.143,A -85,B 0,C 180,E1 -10921.558,E2 -10921.558} C_VEL
LIN {X 0,Y 404.185,Z 67.134,A -85,B 0,C 180,E1 -10925.016,E2 -10925.016} C_VEL
LIN {X 0,Y 404.159,Z 67.137,A -85,B 0,C 180,E1 -10928.756,E2 -10928.756} C_VEL
LIN {X 0,Y 404.124,Z 67.149,A -85,B 0,C 180,E1 -10931.6,E2 -10931.6} C_VEL
LIN {X 0,Y 404.145,Z 67.139,A -85,B 0,C 180,E1 -10934.522,E2 -10934.522} C_VEL
LIN {X 0,Y 404.135,Z 67.146,A -85,B 0,C 180,E1 -10937.295,E2 -10937.295} C_VEL
LIN {X 0,Y 404.168,Z 67.137,A -85,B 0,C 180,E1 -10939.955,E2 -10939.955} C_VEL
LIN {X 0,Y 404.135,Z 67.146,A -85,B 0,C 180,E1 -10943.125,E2 -10943.125} C_VEL
LIN {X 0,Y 404.144,Z 67.139,A -85,B 0,C 180,E1 -10946.188,E2 -10946.188} C_VEL
LIN {X 0,Y 404.145,Z 67.14,A -85,B 0,C 180,E1 -10949.715,E2 -10949.715} C_VEL
LIN {X 0,Y 404.195,Z 67.138,A -85,B 0,C 180,E1 -10953.123,E2 -10953.123} C_VEL
LIN {X 0,Y 404.176,Z 67.137,A -85,B 0,C 180,E1 -10955.334,E2 -10955.334} C_VEL
LIN {X 0,Y 404.138,Z 67.145,A -85,B 0,C 180,E1 -10958.581,E2 -10958.581} C_VEL
LIN {X 0,Y 404.204,Z 67.132,A -85,B 0,C 180,E1 -10961.762,E2 -10961.762} C_VEL
LIN {X 0,Y 404.205,Z 67.135,A -85,B 0,C 180,E1 -10964.882,E2 -10964.882} C_VEL
LIN {X 0,Y 404.255,Z 67.127,A -85,B 0,C 180,E1 -10967.959,E2 -10967.959} C_VEL
LIN {X 0,Y 404.404,Z 67.111,A -85,B 0,C 180,E1 -10972.129,E2 -10972.129} C_VEL
LIN {X 0,Y 404.419,Z 67.109,A -85,B 0,C 180,E1 -10974.015,E2 -10974.015} C_VEL
LIN {X 0,Y 404.477,Z 67.103,A -85,B 0,C 180,E1 -10978.009,E2 -10978.009} C_VEL
LIN {X 0,Y 404.607,Z 67.088,A -85,B 0,C 180,E1 -10980,E2 -10980} C_VEL
LIN {X 0,Y 404.409,Z 67.106,A -85,B 0,C 180,E1 -10982.989,E2 -10982.989} C_VEL
LIN {X 0,Y 404.371,Z 67.112,A -85,B 0,C 180,E1 -10986.509,E2 -10986.509} C_VEL
LIN {X 0,Y 404.265,Z 67.124,A -85,B 0,C 180,E1 -10989.002,E2 -10989.002} C_VEL
LIN {X 0,Y 404.256,Z 67.129,A -85,B 0,C 180,E1 -10992.042,E2 -10992.042} C_VEL
LIN {X 0,Y 404.205,Z 67.133,A -85,B 0,C 180,E1 -10995.118,E2 -10995.118} C_VEL
LIN {X 0,Y 404.208,Z 67.132,A -85,B 0,C 180,E1 -10998.239,E2 -10998.239} C_VEL
LIN {X 0,Y 404.16,Z 67.144,A -85,B 0,C 180,E1 -11001.419,E2 -11001.419} C_VEL
LIN {X 0,Y 404.172,Z 67.137,A -85,B 0,C 180,E1 -11004.666,E2 -11004.666} C_VEL
LIN {X 0,Y 404.195,Z 67.133,A -85,B 0,C 180,E1 -11008,E2 -11008} C_VEL
LIN {X 0,Y 404.14,Z 67.142,A -85,B 0,C 180,E1 -11011.558,E2 -11011.558} C_VEL
LIN {X 0,Y 404.184,Z 67.141,A -85,B 0,C 180,E1 -11015.017,E2 -11015.017} C_VEL
LIN {X 0,Y 404.138,Z 67.146,A -85,B 0,C 180,E1 -11018.759,E2 -11018.759} C_VEL
LIN {X 0,Y 404.11,Z 67.144,A -85,B 0,C 180,E1 -11021.598,E2 -11021.598} C_VEL
LIN {X 0,Y 404.145,Z 67.144,A -85,B 0,C 180,E1 -11024.522,E2 -11024.522} C_VEL
LIN {X 0,Y 404.134,Z 67.141,A -85,B 0,C 180,E1 -11027.296,E2 -11027.296} C_VEL
LIN {X 0,Y 404.133,Z 67.142,A -85,B 0,C 180,E1 -11029.951,E2 -11029.951} C_VEL
LIN {X 0,Y 404.136,Z 67.141,A -85,B 0,C 180,E1 -11033.126,E2 -11033.126} C_VEL
LIN {X 0,Y 404.147,Z 67.144,A -85,B 0,C 180,E1 -11036.188,E2 -11036.188} C_VEL
LIN {X 0,Y 404.147,Z 67.141,A -85,B 0,C 180,E1 -11039.715,E2 -11039.715} C_VEL
LIN {X 0,Y 404.136,Z 67.14,A -85,B 0,C 180,E1 -11043.119,E2 -11043.119} C_VEL
LIN {X 0,Y 404.156,Z 67.14,A -85,B 0,C 180,E1 -11046.425,E2 -11046.425} C_VEL
LIN {X 0,Y 404.195,Z 67.14,A -85,B 0,C 180,E1 -11049.875,E2 -11049.875} C_VEL
LIN {X 0,Y 404.22,Z 67.132,A -85,B 0,C 180,E1 -11052.993,E2 -11052.993} C_VEL
LIN {X 0,Y 404.261,Z 67.238,A -85,B 0,C 180,E1 -11055.271,E2 -11055.271} C_VEL
LIN {X 0,Y 405.765,Z 76.067,A -85,B 0,C 180,E1 -11057.496,E2 -11057.496} C_VEL
LIN {X 0,Y 405.932,Z 77.723,A -85,B 0,C 180,E1 -11057.84,E2 -11057.84} C_VEL
LIN {X 0,Y 409.634,Z 96.616,A -85,B 0,C 180,E1 -11058.34,E2 -11058.34} C_VEL
LIN {X 0,Y 408.595,Z 184.825,A -85,B 0,C 180,E1 -11059.908,E2 -11059.908} C_VEL
LIN {X 0,Y 408.317,Z 197.766,A -85,B 0,C 180,E1 -11060.339,E2 -11060.339} C_VEL
LIN {X 0,Y 407.821,Z 210.304,A -85,B 0,C 180,E1 -11060.953,E2 -11060.953} C_VEL
LIN {X 0,Y 407.39,Z 221.45,A -85,B 0,C 180,E1 -11061.693,E2 -11061.693} C_VEL
LIN {X 0,Y 406.64,Z 233.001,A -85,B 0,C 180,E1 -11062.677,E2 -11062.677} C_VEL
LIN {X 0,Y 405.925,Z 243.384,A -85,B 0,C 180,E1 -11063.788,E2 -11063.788} C_VEL
LIN {X 0,Y 405.21,Z 253.277,A -85,B 0,C 180,E1 -11065.106,E2 -11065.106} C_VEL
LIN {X 0,Y 404.518,Z 261.777,A -85,B 0,C 180,E1 -11066.514,E2 -11066.514} C_VEL
LIN {X 0,Y 403.956,Z 269.053,A -85,B 0,C 180,E1 -11068.006,E2 -11068.006} C_VEL
LIN {X 0,Y 403.817,Z 271.416,A -85,B 0,C 180,E1 -11068.576,E2 -11068.576} C_VEL
LIN {X 0,Y 402.91,Z 274.268,A -85,B 0,C 180,E1 -11069.305,E2 -11069.305} C_VEL
LIN {X 0,Y 399.783,Z 278.396,A -85,B 0,C 180,E1 -11070.513,E2 -11070.513} C_VEL
LIN {X 0,Y 396.761,Z 281.876,A -85,B 0,C 180,E1 -11071.78,E2 -11071.78} C_VEL
LIN {X 0,Y 396.027,Z 283.536,A -85,B 0,C 180,E1 -11072.59,E2 -11072.59} C_VEL
LIN {X 0,Y 395.876,Z 285.995,A -85,B 0,C 180,E1 -11074.072,E2 -11074.072} C_VEL
LIN {X 0,Y 395.902,Z 287.134,A -85,B 0,C 180,E1 -11075.093,E2 -11075.093} C_VEL
LIN {X 0,Y 395.948,Z 287.925,A -85,B 0,C 180,E1 -11076.281,E2 -11076.281} C_VEL
LIN {X 0,Y 395.837,Z 288.142,A -85,B 0,C 180,E1 -11078.166,E2 -11078.166} C_VEL
LIN {X 0,Y 395.84,Z 287.692,A -85,B 0,C 180,E1 -11079.195,E2 -11079.195} C_VEL
LIN {X 0,Y 396.046,Z 285.534,A -85,B 0,C 180,E1 -11081.257,E2 -11081.257} C_VEL
LIN {X 0,Y 396.352,Z 282.878,A -85,B 0,C 180,E1 -11082.773,E2 -11082.773} C_VEL
LIN {X 0,Y 396.672,Z 279.049,A -85,B 0,C 180,E1 -11084.362,E2 -11084.362} C_VEL
LIN {X 0,Y 397.224,Z 274.132,A -85,B 0,C 180,E1 -11085.917,E2 -11085.917} C_VEL
LIN {X 0,Y 397.861,Z 267.907,A -85,B 0,C 180,E1 -11087.476,E2 -11087.476} C_VEL
LIN {X 0,Y 398.614,Z 260.083,A -85,B 0,C 180,E1 -11089.037,E2 -11089.037} C_VEL
LIN {X 0,Y 399.472,Z 252.039,A -85,B 0,C 180,E1 -11090.333,E2 -11090.333} C_VEL
LIN {X 0,Y 400.398,Z 242.174,A -85,B 0,C 180,E1 -11091.63,E2 -11091.63} C_VEL
LIN {X 0,Y 401.242,Z 232.456,A -85,B 0,C 180,E1 -11092.665,E2 -11092.665} C_VEL
LIN {X 0,Y 402.102,Z 221.953,A -85,B 0,C 180,E1 -11093.567,E2 -11093.567} C_VEL
LIN {X 0,Y 402.894,Z 210.399,A -85,B 0,C 180,E1 -11094.338,E2 -11094.338} C_VEL
LIN {X 0,Y 403.522,Z 197.056,A -85,B 0,C 180,E1 -11094.992,E2 -11094.992} C_VEL
LIN {X 0,Y 404.014,Z 184.544,A -85,B 0,C 180,E1 -11095.395,E2 -11095.395} C_VEL
LIN {X 0,Y 405.244,Z 98.825,A -85,B 0,C 180,E1 -11096.955,E2 -11096.955} C_VEL
LIN {X 0,Y 401.355,Z 83.721,A -85,B 0,C 180,E1 -11097.475,E2 -11097.475} C_VEL
LIN {X 0,Y 399.169,Z 78.045,A -85,B 0,C 180,E1 -11097.738,E2 -11097.738} C_VEL
LIN {X 0,Y 397.113,Z 68.021,A -85,B 0,C 180,E1 -11100.487,E2 -11100.487} C_VEL
LIN {X 0,Y 397.1,Z 68.025,A -85,B 0,C 180,E1 -11103.713,E2 -11103.713} C_VEL
LIN {X 0,Y 397.09,Z 68.018,A -85,B 0,C 180,E1 -11107.207,E2 -11107.207} C_VEL
LIN {X 0,Y 397.058,Z 68.026,A -85,B 0,C 180,E1 -11110.437,E2 -11110.437} C_VEL
LIN {X 0,Y 397.09,Z 68.017,A -85,B 0,C 180,E1 -11113.651,E2 -11113.651} C_VEL
LIN {X 0,Y 397.094,Z 68.02,A -85,B 0,C 180,E1 -11116.523,E2 -11116.523} C_VEL
LIN {X 0,Y 397.087,Z 68.02,A -85,B 0,C 180,E1 -11120.419,E2 -11120.419} C_VEL
LIN {X 0,Y 397.094,Z 68.021,A -85,B 0,C 180,E1 -11123.004,E2 -11123.004} C_VEL
LIN {X 0,Y 397.113,Z 68.018,A -85,B 0,C 180,E1 -11126.726,E2 -11126.726} C_VEL
LIN {X 0,Y 397.116,Z 68.016,A -85,B 0,C 180,E1 -11130.295,E2 -11130.295} C_VEL
LIN {X 0,Y 397.073,Z 68.022,A -85,B 0,C 180,E1 -11133.737,E2 -11133.737} C_VEL
LIN {X 0,Y 397.102,Z 68.015,A -85,B 0,C 180,E1 -11137.085,E2 -11137.085} C_VEL
LIN {X 0,Y 397.15,Z 68.013,A -85,B 0,C 180,E1 -11140.353,E2 -11140.353} C_VEL
LIN {X 0,Y 397.167,Z 68.007,A -85,B 0,C 180,E1 -11143.553,E2 -11143.553} C_VEL
LIN {X 0,Y 397.233,Z 68,A -85,B 0,C 180,E1 -11146.703,E2 -11146.703} C_VEL
LIN {X 0,Y 397.217,Z 68.002,A -85,B 0,C 180,E1 -11149.809,E2 -11149.809} C_VEL
LIN {X 0,Y 397.292,Z 67.988,A -85,B 0,C 180,E1 -11152.887,E2 -11152.887} C_VEL
LIN {X 0,Y 397.232,Z 68,A -85,B 0,C 180,E1 -11154.925,E2 -11154.925} C_VEL
LIN {X 0,Y 397.447,Z 67.978,A -85,B 0,C 180,E1 -11157.973,E2 -11157.973} C_VEL
LIN {X 0,Y 397.443,Z 67.977,A -85,B 0,C 180,E1 -11162.027,E2 -11162.027} C_VEL
LIN {X 0,Y 397.332,Z 67.983,A -85,B 0,C 180,E1 -11166.092,E2 -11166.092} C_VEL
LIN {X 0,Y 397.237,Z 68.001,A -85,B 0,C 180,E1 -11169.162,E2 -11169.162} C_VEL
LIN {X 0,Y 397.222,Z 67.999,A -85,B 0,C 180,E1 -11172.258,E2 -11172.258} C_VEL
LIN {X 0,Y 397.179,Z 68.011,A -85,B 0,C 180,E1 -11175.392,E2 -11175.392} C_VEL
LIN {X 0,Y 397.159,Z 68.008,A -85,B 0,C 180,E1 -11178.573,E2 -11178.573} C_VEL
LIN {X 0,Y 397.099,Z 68.012,A -85,B 0,C 180,E1 -11181.818,E2 -11181.818} C_VEL
LIN {X 0,Y 397.157,Z 68.016,A -85,B 0,C 180,E1 -11185.131,E2 -11185.131} C_VEL
LIN {X 0,Y 397.164,Z 68.01,A -85,B 0,C 180,E1 -11187.776,E2 -11187.776} C_VEL
LIN {X 0,Y 397.081,Z 68.02,A -85,B 0,C 180,E1 -11190.882,E2 -11190.882} C_VEL
LIN {X 0,Y 397.128,Z 68.015,A -85,B 0,C 180,E1 -11194.493,E2 -11194.493} C_VEL
LIN {X 0,Y 397.104,Z 68.013,A -85,B 0,C 180,E1 -11198.275,E2 -11198.275} C_VEL
LIN {X 0,Y 397.091,Z 68.02,A -85,B 0,C 180,E1 -11200.908,E2 -11200.908} C_VEL
LIN {X 0,Y 397.103,Z 68.018,A -85,B 0,C 180,E1 -11203.648,E2 -11203.648} C_VEL
LIN {X 0,Y 397.104,Z 68.018,A -85,B 0,C 180,E1 -11206.521,E2 -11206.521} C_VEL
LIN {X 0,Y 397.117,Z 68.016,A -85,B 0,C 180,E1 -11210.423,E2 -11210.423} C_VEL
LIN {X 0,Y 397.11,Z 68.015,A -85,B 0,C 180,E1 -11214.265,E2 -11214.265} C_VEL
LIN {X 0,Y 397.117,Z 68.022,A -85,B 0,C 180,E1 -11216.727,E2 -11216.727} C_VEL
LIN {X 0,Y 397.139,Z 68.12,A -85,B 0,C 180,E1 -11220.169,E2 -11220.169} C_VEL
LIN {X 0,Y 399.926,Z 80.359,A -85,B 0,C 180,E1 -11223.055,E2 -11223.055} C_VEL
LIN {X 0,Y 401.18,Z 87.135,A -85,B 0,C 180,E1 -11224.583,E2 -11224.583} C_VEL
LIN {X 0,Y 400.114,Z 100.273,A -85,B 0,C 180,E1 -11227.267,E2 -11227.267} C_VEL
LIN {X 0,Y 399.305,Z 110.494,A -85,B 0,C 180,E1 -11229.331,E2 -11229.331} C_VEL
LIN {X 0,Y 404.042,Z 136.984,A -85,B 0,C 180,E1 -11230.115,E2 -11230.115} C_VEL
LIN {X 0,Y 404.683,Z 143.337,A -85,B 0,C 180,E1 -11230.271,E2 -11230.271} C_VEL
LIN {X 0,Y 403.56,Z 219.827,A -85,B 0,C 180,E1 -11231.67,E2 -11231.67} C_VEL
LIN {X 0,Y 402.87,Z 233.49,A -85,B 0,C 180,E1 -11232.126,E2 -11232.126} C_VEL
LIN {X 0,Y 401.948,Z 246.411,A -85,B 0,C 180,E1 -11232.773,E2 -11232.773} C_VEL
LIN {X 0,Y 401.025,Z 258.163,A -85,B 0,C 180,E1 -11233.585,E2 -11233.585} C_VEL
LIN {X 0,Y 399.98,Z 269.502,A -85,B 0,C 180,E1 -11234.588,E2 -11234.588} C_VEL
LIN {X 0,Y 398.953,Z 279.749,A -85,B 0,C 180,E1 -11235.722,E2 -11235.722} C_VEL
LIN {X 0,Y 398.169,Z 288.975,A -85,B 0,C 180,E1 -11236.994,E2 -11236.994} C_VEL
LIN {X 0,Y 397.209,Z 297.961,A -85,B 0,C 180,E1 -11238.518,E2 -11238.518} C_VEL
LIN {X 0,Y 396.599,Z 305.219,A -85,B 0,C 180,E1 -11240.05,E2 -11240.05} C_VEL
LIN {X 0,Y 396.226,Z 310.139,A -85,B 0,C 180,E1 -11241.328,E2 -11241.328} C_VEL
LIN {X 0,Y 395.948,Z 314.934,A -85,B 0,C 180,E1 -11242.862,E2 -11242.862} C_VEL
LIN {X 0,Y 395.794,Z 318.294,A -85,B 0,C 180,E1 -11244.239,E2 -11244.239} C_VEL
LIN {X 0,Y 395.777,Z 321.305,A -85,B 0,C 180,E1 -11245.927,E2 -11245.927} C_VEL
LIN {X 0,Y 395.858,Z 323.448,A -85,B 0,C 180,E1 -11247.965,E2 -11247.965} C_VEL
LIN {X 0,Y 395.835,Z 323.879,A -85,B 0,C 180,E1 -11248.982,E2 -11248.982} C_VEL
LIN {X 0,Y 395.827,Z 323.921,A -85,B 0,C 180,E1 -11250,E2 -11250} C_VEL
LIN {X 0,Y 395.883,Z 322.841,A -85,B 0,C 180,E1 -11252.034,E2 -11252.034} C_VEL
LIN {X 0,Y 395.811,Z 321.652,A -85,B 0,C 180,E1 -11253.053,E2 -11253.053} C_VEL
LIN {X 0,Y 395.843,Z 319.108,A -85,B 0,C 180,E1 -11254.582,E2 -11254.582} C_VEL
LIN {X 0,Y 395.787,Z 315.531,A -85,B 0,C 180,E1 -11256.116,E2 -11256.116} C_VEL
LIN {X 0,Y 396.027,Z 310.845,A -85,B 0,C 180,E1 -11257.648,E2 -11257.648} C_VEL
LIN {X 0,Y 396.363,Z 303.76,A -85,B 0,C 180,E1 -11259.44,E2 -11259.44} C_VEL
LIN {X 0,Y 396.784,Z 296.079,A -85,B 0,C 180,E1 -11260.976,E2 -11260.976} C_VEL
LIN {X 0,Y 397.416,Z 288.225,A -85,B 0,C 180,E1 -11262.252,E2 -11262.252} C_VEL
LIN {X 0,Y 398.189,Z 278.192,A -85,B 0,C 180,E1 -11263.576,E2 -11263.576} C_VEL
LIN {X 0,Y 398.786,Z 267.94,A -85,B 0,C 180,E1 -11264.675,E2 -11264.675} C_VEL
LIN {X 0,Y 399.683,Z 256.013,A -85,B 0,C 180,E1 -11265.685,E2 -11265.685} C_VEL
LIN {X 0,Y 400.466,Z 243.201,A -85,B 0,C 180,E1 -11266.504,E2 -11266.504} C_VEL
LIN {X 0,Y 401.103,Z 231.128,A -85,B 0,C 180,E1 -11267.067,E2 -11267.067} C_VEL
LIN {X 0,Y 401.559,Z 217.858,A -85,B 0,C 180,E1 -11267.473,E2 -11267.473} C_VEL
LIN {X 0,Y 402.322,Z 139.804,A -85,B 0,C 180,E1 -11268.878,E2 -11268.878} C_VEL
LIN {X 0,Y 398.339,Z 110.816,A -85,B 0,C 180,E1 -11269.586,E2 -11269.586} C_VEL
LIN {X 0,Y 399.58,Z 91.925,A -85,B 0,C 180,E1 -11273.312,E2 -11273.312} C_VEL
LIN {X 0,Y 400.121,Z 83.78,A -85,B 0,C 180,E1 -11274.932,E2 -11274.932} C_VEL
LIN {X 0,Y 398.176,Z 72.675,A -85,B 0,C 180,E1 -11277.317,E2 -11277.317} C_VEL
LIN {X 0,Y 397.178,Z 68.009,A -85,B 0,C 180,E1 -11278.395,E2 -11278.395} C_VEL
LIN {X 0,Y 397.079,Z 68.024,A -85,B 0,C 180,E1 -11282.071,E2 -11282.071} C_VEL
LIN {X 0,Y 397.12,Z 68.018,A -85,B 0,C 180,E1 -11285.503,E2 -11285.503} C_VEL
LIN {X 0,Y 397.134,Z 68.013,A -85,B 0,C 180,E1 -11288.862,E2 -11288.862} C_VEL
LIN {X 0,Y 397.069,Z 68.021,A -85,B 0,C 180,E1 -11292.267,E2 -11292.267} C_VEL
LIN {X 0,Y 397.086,Z 68.021,A -85,B 0,C 180,E1 -11295.069,E2 -11295.069} C_VEL
LIN {X 0,Y 397.065,Z 68.022,A -85,B 0,C 180,E1 -11298.021,E2 -11298.021} C_VEL
LIN {X 0,Y 397.127,Z 68.018,A -85,B 0,C 180,E1 -11301.139,E2 -11301.139} C_VEL
LIN {X 0,Y 397.118,Z 68.015,A -85,B 0,C 180,E1 -11304.497,E2 -11304.497} C_VEL
LIN {X 0,Y 397.077,Z 68.02,A -85,B 0,C 180,E1 -11307.928,E2 -11307.928} C_VEL
LIN {X 0,Y 397.121,Z 68.016,A -85,B 0,C 180,E1 -11311.456,E2 -11311.456} C_VEL
LIN {X 0,Y 397.152,Z 68.013,A -85,B 0,C 180,E1 -11314.488,E2 -11314.488} C_VEL
LIN {X 0,Y 397.108,Z 68.019,A -85,B 0,C 180,E1 -11317.086,E2 -11317.086} C_VEL
LIN {X 0,Y 397.146,Z 68.014,A -85,B 0,C 180,E1 -11320.353,E2 -11320.353} C_VEL
LIN {X 0,Y 397.166,Z 68.009,A -85,B 0,C 180,E1 -11323.553,E2 -11323.553} C_VEL
LIN {X 0,Y 397.228,Z 68.005,A -85,B 0,C 180,E1 -11326.703,E2 -11326.703} C_VEL
LIN {X 0,Y 397.216,Z 68.003,A -85,B 0,C 180,E1 -11329.809,E2 -11329.809} C_VEL
LIN {X 0,Y 397.349,Z 67.987,A -85,B 0,C 180,E1 -11332.888,E2 -11332.888} C_VEL
LIN {X 0,Y 397.251,Z 67.999,A -85,B 0,C 180,E1 -11334.925,E2 -11334.925} C_VEL
LIN {X 0,Y 397.446,Z 67.978,A -85,B 0,C 180,E1 -11337.973,E2 -11337.973} C_VEL
LIN {X 0,Y 397.576,Z 67.963,A -85,B 0,C 180,E1 -11340,E2 -11340} C_VEL
LIN {X 0,Y 397.369,Z 67.983,A -85,B 0,C 180,E1 -11343.042,E2 -11343.042} C_VEL
LIN {X 0,Y 397.325,Z 67.99,A -85,B 0,C 180,E1 -11346.502,E2 -11346.502} C_VEL
LIN {X 0,Y 397.235,Z 68.001,A -85,B 0,C 180,E1 -11349.163,E2 -11349.163} C_VEL
LIN {X 0,Y 397.219,Z 68.003,A -85,B 0,C 180,E1 -11352.258,E2 -11352.258} C_VEL
LIN {X 0,Y 397.178,Z 68.011,A -85,B 0,C 180,E1 -11355.392,E2 -11355.392} C_VEL
LIN {X 0,Y 397.16,Z 68.009,A -85,B 0,C 180,E1 -11358.574,E2 -11358.574} C_VEL
LIN {X 0,Y 397.109,Z 68.018,A -85,B 0,C 180,E1 -11361.818,E2 -11361.818} C_VEL
LIN {X 0,Y 397.151,Z 68.015,A -85,B 0,C 180,E1 -11365.512,E2 -11365.512} C_VEL
LIN {X 0,Y 397.122,Z 68.015,A -85,B 0,C 180,E1 -11368.544,E2 -11368.544} C_VEL
LIN {X 0,Y 397.079,Z 68.019,A -85,B 0,C 180,E1 -11372.072,E2 -11372.072} C_VEL
LIN {X 0,Y 397.119,Z 68.016,A -85,B 0,C 180,E1 -11375.504,E2 -11375.504} C_VEL
LIN {X 0,Y 397.096,Z 68.024,A -85,B 0,C 180,E1 -11378.856,E2 -11378.856} C_VEL
LIN {X 0,Y 397.057,Z 68.024,A -85,B 0,C 180,E1 -11382.269,E2 -11382.269} C_VEL
LIN {X 0,Y 397.087,Z 68.021,A -85,B 0,C 180,E1 -11385.069,E2 -11385.069} C_VEL
LIN {X 0,Y 397.063,Z 68.023,A -85,B 0,C 180,E1 -11388.022,E2 -11388.022} C_VEL
LIN {X 0,Y 397.101,Z 68.017,A -85,B 0,C 180,E1 -11391.145,E2 -11391.145} C_VEL
LIN {X 0,Y 397.121,Z 68.02,A -85,B 0,C 180,E1 -11394.497,E2 -11394.497} C_VEL
LIN {X 0,Y 397.081,Z 68.022,A -85,B 0,C 180,E1 -11397.929,E2 -11397.929} C_VEL
LIN {X 0,Y 397.121,Z 68.02,A -85,B 0,C 180,E1 -11400.296,E2 -11400.296} C_VEL
LIN {X 0,Y 397.094,Z 68.021,A -85,B 0,C 180,E1 -11403.739,E2 -11403.739} C_VEL
LIN {X 0,Y 397.104,Z 68.016,A -85,B 0,C 180,E1 -11407.086,E2 -11407.086} C_VEL
LIN {X 0,Y 397.151,Z 68.012,A -85,B 0,C 180,E1 -11410.353,E2 -11410.353} C_VEL
LIN {X 0,Y 397.17,Z 68.012,A -85,B 0,C 180,E1 -11413.554,E2 -11413.554} C_VEL
LIN {X 0,Y 397.201,Z 68.126,A -85,B 0,C 180,E1 -11415.069,E2 -11415.069} C_VEL
LIN {X 0,Y 398.849,Z 77.717,A -85,B 0,C 180,E1 -11417.518,E2 -11417.518} C_VEL
LIN {X 0,Y 402.268,Z 94.004,A -85,B 0,C 180,E1 -11417.978,E2 -11417.978} C_VEL
LIN {X 0,Y 402.939,Z 99.693,A -85,B 0,C 180,E1 -11418.111,E2 -11418.111} C_VEL
LIN {X 0,Y 401.754,Z 184.756,A -85,B 0,C 180,E1 -11419.639,E2 -11419.639} C_VEL
LIN {X 0,Y 401.465,Z 197.826,A -85,B 0,C 180,E1 -11420.077,E2 -11420.077} C_VEL
LIN {X 0,Y 400.979,Z 209.871,A -85,B 0,C 180,E1 -11420.67,E2 -11420.67} C_VEL
LIN {X 0,Y 400.522,Z 221.215,A -85,B 0,C 180,E1 -11421.423,E2 -11421.423} C_VEL
LIN {X 0,Y 399.759,Z 232.89,A -85,B 0,C 180,E1 -11422.424,E2 -11422.424} C_VEL
LIN {X 0,Y 399.009,Z 243.347,A -85,B 0,C 180,E1 -11423.553,E2 -11423.553} C_VEL
LIN {X 0,Y 398.337,Z 251.904,A -85,B 0,C 180,E1 -11424.686,E2 -11424.686} C_VEL
LIN {X 0,Y 397.69,Z 259.792,A -85,B 0,C 180,E1 -11425.947,E2 -11425.947} C_VEL
LIN {X 0,Y 397.071,Z 267.529,A -85,B 0,C 180,E1 -11427.464,E2 -11427.464} C_VEL
LIN {X 0,Y 396.58,Z 273.719,A -85,B 0,C 180,E1 -11428.985,E2 -11428.985} C_VEL
LIN {X 0,Y 396.228,Z 278.648,A -85,B 0,C 180,E1 -11430.508,E2 -11430.508} C_VEL
LIN {X 0,Y 396.091,Z 282.461,A -85,B 0,C 180,E1 -11432.034,E2 -11432.034} C_VEL
LIN {X 0,Y 396.027,Z 283.536,A -85,B 0,C 180,E1 -11432.59,E2 -11432.59} C_VEL
LIN {X 0,Y 395.313,Z 285.082,A -85,B 0,C 180,E1 -11433.411,E2 -11433.411} C_VEL
LIN {X 0,Y 392.41,Z 286.951,A -85,B 0,C 180,E1 -11434.761,E2 -11434.761} C_VEL
LIN {X 0,Y 389.965,Z 287.987,A -85,B 0,C 180,E1 -11435.865,E2 -11435.865} C_VEL
LIN {X 0,Y 388.827,Z 288.454,A -85,B 0,C 180,E1 -11436.868,E2 -11436.868} C_VEL
LIN {X 0,Y 388.797,Z 288.446,A -85,B 0,C 180,E1 -11437.014,E2 -11437.014} C_VEL
LIN {X 0,Y 388.767,Z 288.45,A -85,B 0,C 180,E1 -11438.316,E2 -11438.316} C_VEL
LIN {X 0,Y 388.768,Z 287.948,A -85,B 0,C 180,E1 -11439.364,E2 -11439.364} C_VEL
LIN {X 0,Y 389.001,Z 285.736,A -85,B 0,C 180,E1 -11441.463,E2 -11441.463} C_VEL
LIN {X 0,Y 389.296,Z 283.301,A -85,B 0,C 180,E1 -11442.87,E2 -11442.87} C_VEL
LIN {X 0,Y 389.674,Z 279.135,A -85,B 0,C 180,E1 -11444.626,E2 -11444.626} C_VEL
LIN {X 0,Y 390.253,Z 274.154,A -85,B 0,C 180,E1 -11446.209,E2 -11446.209} C_VEL
LIN {X 0,Y 390.946,Z 267.856,A -85,B 0,C 180,E1 -11447.795,E2 -11447.795} C_VEL
LIN {X 0,Y 391.776,Z 259.911,A -85,B 0,C 180,E1 -11449.383,E2 -11449.383} C_VEL
LIN {X 0,Y 392.701,Z 251.768,A -85,B 0,C 180,E1 -11450.699,E2 -11450.699} C_VEL
LIN {X 0,Y 393.676,Z 241.785,A -85,B 0,C 180,E1 -11452.018,E2 -11452.018} C_VEL
LIN {X 0,Y 394.707,Z 230.482,A -85,B 0,C 180,E1 -11453.201,E2 -11453.201} C_VEL
LIN {X 0,Y 395.593,Z 219.335,A -85,B 0,C 180,E1 -11454.118,E2 -11454.118} C_VEL
LIN {X 0,Y 396.47,Z 206.926,A -85,B 0,C 180,E1 -11454.898,E2 -11454.898} C_VEL
LIN {X 0,Y 397.047,Z 194.349,A -85,B 0,C 180,E1 -11455.464,E2 -11455.464} C_VEL
LIN {X 0,Y 397.456,Z 180.44,A -85,B 0,C 180,E1 -11455.856,E2 -11455.856} C_VEL
LIN {X 0,Y 398.677,Z 100.042,A -85,B 0,C 180,E1 -11457.326,E2 -11457.326} C_VEL
LIN {X 0,Y 395.226,Z 86.527,A -85,B 0,C 180,E1 -11457.802,E2 -11457.802} C_VEL
LIN {X 0,Y 392.063,Z 78.36,A -85,B 0,C 180,E1 -11458.188,E2 -11458.188} C_VEL
LIN {X 0,Y 390.051,Z 68.901,A -85,B 0,C 180,E1 -11460.824,E2 -11460.824} C_VEL
LIN {X 0,Y 390.073,Z 68.898,A -85,B 0,C 180,E1 -11464.025,E2 -11464.025} C_VEL
LIN {X 0,Y 390.038,Z 68.896,A -85,B 0,C 180,E1 -11467.781,E2 -11467.781} C_VEL
LIN {X 0,Y 390.019,Z 68.902,A -85,B 0,C 180,E1 -11470.814,E2 -11470.814} C_VEL
LIN {X 0,Y 390.047,Z 68.891,A -85,B 0,C 180,E1 -11473.884,E2 -11473.884} C_VEL
LIN {X 0,Y 390.05,Z 68.897,A -85,B 0,C 180,E1 -11476.788,E2 -11476.788} C_VEL
LIN {X 0,Y 390.012,Z 68.904,A -85,B 0,C 180,E1 -11479.554,E2 -11479.554} C_VEL
LIN {X 0,Y 390.038,Z 68.898,A -85,B 0,C 180,E1 -11482.451,E2 -11482.451} C_VEL
LIN {X 0,Y 390.065,Z 68.896,A -85,B 0,C 180,E1 -11486.044,E2 -11486.044} C_VEL
LIN {X 0,Y 390.043,Z 68.898,A -85,B 0,C 180,E1 -11489.871,E2 -11489.871} C_VEL
LIN {X 0,Y 390.029,Z 68.898,A -85,B 0,C 180,E1 -11493.225,E2 -11493.225} C_VEL
LIN {X 0,Y 390.062,Z 68.893,A -85,B 0,C 180,E1 -11496.767,E2 -11496.767} C_VEL
LIN {X 0,Y 390.107,Z 68.889,A -85,B 0,C 180,E1 -11499.983,E2 -11499.983} C_VEL
LIN {X 0,Y 390.14,Z 68.884,A -85,B 0,C 180,E1 -11503.248,E2 -11503.248} C_VEL
LIN {X 0,Y 390.198,Z 68.878,A -85,B 0,C 180,E1 -11506.561,E2 -11506.561} C_VEL
LIN {X 0,Y 390.168,Z 68.879,A -85,B 0,C 180,E1 -11509.623,E2 -11509.623} C_VEL
LIN {X 0,Y 390.246,Z 68.866,A -85,B 0,C 180,E1 -11512.758,E2 -11512.758} C_VEL
LIN {X 0,Y 390.203,Z 68.876,A -85,B 0,C 180,E1 -11514.833,E2 -11514.833} C_VEL
LIN {X 0,Y 390.414,Z 68.854,A -85,B 0,C 180,E1 -11517.937,E2 -11517.937} C_VEL
LIN {X 0,Y 390.41,Z 68.853,A -85,B 0,C 180,E1 -11522.063,E2 -11522.063} C_VEL
LIN {X 0,Y 390.286,Z 68.861,A -85,B 0,C 180,E1 -11526.202,E2 -11526.202} C_VEL
LIN {X 0,Y 390.195,Z 68.879,A -85,B 0,C 180,E1 -11529.329,E2 -11529.329} C_VEL
LIN {X 0,Y 390.174,Z 68.876,A -85,B 0,C 180,E1 -11532.483,E2 -11532.483} C_VEL
LIN {X 0,Y 390.14,Z 68.884,A -85,B 0,C 180,E1 -11535.677,E2 -11535.677} C_VEL
LIN {X 0,Y 390.104,Z 68.888,A -85,B 0,C 180,E1 -11538.922,E2 -11538.922} C_VEL
LIN {X 0,Y 390.042,Z 68.889,A -85,B 0,C 180,E1 -11542.234,E2 -11542.234} C_VEL
LIN {X 0,Y 390.12,Z 68.886,A -85,B 0,C 180,E1 -11545.743,E2 -11545.743} C_VEL
LIN {X 0,Y 390.061,Z 68.9,A -85,B 0,C 180,E1 -11549.109,E2 -11549.109} C_VEL
LIN {X 0,Y 390.046,Z 68.899,A -85,B 0,C 180,E1 -11552.721,E2 -11552.721} C_VEL
LIN {X 0,Y 390.058,Z 68.88,A -85,B 0,C 180,E1 -11555.825,E2 -11555.825} C_VEL
LIN {X 0,Y 390.071,Z 68.897,A -85,B 0,C 180,E1 -11559.218,E2 -11559.218} C_VEL
LIN {X 0,Y 390.045,Z 68.9,A -85,B 0,C 180,E1 -11562.374,E2 -11562.374} C_VEL
LIN {X 0,Y 390.046,Z 68.896,A -85,B 0,C 180,E1 -11565.354,E2 -11565.354} C_VEL
LIN {X 0,Y 390.034,Z 68.898,A -85,B 0,C 180,E1 -11568.187,E2 -11568.187} C_VEL
LIN {X 0,Y 390.094,Z 68.892,A -85,B 0,C 180,E1 -11570.908,E2 -11570.908} C_VEL
LIN {X 0,Y 390.087,Z 68.889,A -85,B 0,C 180,E1 -11574.793,E2 -11574.793} C_VEL
LIN {X 0,Y 390.026,Z 68.908,A -85,B 0,C 180,E1 -11578.495,E2 -11578.495} C_VEL
LIN {X 0,Y 390.056,Z 68.926,A -85,B 0,C 180,E1 -11579.767,E2 -11579.767} C_VEL
LIN {X 0,Y 392.748,Z 80.47,A -85,B 0,C 180,E1 -11582.561,E2 -11582.561} C_VEL
LIN {X 0,Y 394.255,Z 88.373,A -85,B 0,C 180,E1 -11584.387,E2 -11584.387} C_VEL
LIN {X 0,Y 393.782,Z 94.936,A -85,B 0,C 180,E1 -11585.764,E2 -11585.764} C_VEL
LIN {X 0,Y 392.48,Z 110.221,A -85,B 0,C 180,E1 -11588.908,E2 -11588.908} C_VEL
LIN {X 0,Y 397.326,Z 137.009,A -85,B 0,C 180,E1 -11589.723,E2 -11589.723} C_VEL
LIN {X 0,Y 398.109,Z 143.959,A -85,B 0,C 180,E1 -11589.903,E2 -11589.903} C_VEL
LIN {X 0,Y 396.946,Z 218.869,A -85,B 0,C 180,E1 -11591.29,E2 -11591.29} C_VEL
LIN {X 0,Y 396.296,Z 231.914,A -85,B 0,C 180,E1 -11591.719,E2 -11591.719} C_VEL
LIN {X 0,Y 395.379,Z 244.658,A -85,B 0,C 180,E1 -11592.344,E2 -11592.344} C_VEL
LIN {X 0,Y 394.389,Z 256.791,A -85,B 0,C 180,E1 -11593.167,E2 -11593.167} C_VEL
LIN {X 0,Y 393.244,Z 268.322,A -85,B 0,C 180,E1 -11594.184,E2 -11594.184} C_VEL
LIN {X 0,Y 392.162,Z 278.723,A -85,B 0,C 180,E1 -11595.336,E2 -11595.336} C_VEL
LIN {X 0,Y 391.39,Z 287.242,A -85,B 0,C 180,E1 -11596.5,E2 -11596.5} C_VEL
LIN {X 0,Y 390.592,Z 295.12,A -85,B 0,C 180,E1 -11597.794,E2 -11597.794} C_VEL
LIN {X 0,Y 389.776,Z 302.837,A -85,B 0,C 180,E1 -11599.349,E2 -11599.349} C_VEL
LIN {X 0,Y 389.177,Z 309.963,A -85,B 0,C 180,E1 -11601.17,E2 -11601.17} C_VEL
LIN {X 0,Y 388.896,Z 314.728,A -85,B 0,C 180,E1 -11602.732,E2 -11602.732} C_VEL
LIN {X 0,Y 388.749,Z 317.551,A -85,B 0,C 180,E1 -11603.89,E2 -11603.89} C_VEL
LIN {X 0,Y 388.699,Z 321.042,A -85,B 0,C 180,E1 -11605.852,E2 -11605.852} C_VEL
LIN {X 0,Y 388.671,Z 322.3,A -85,B 0,C 180,E1 -11606.89,E2 -11606.89} C_VEL
LIN {X 0,Y 388.756,Z 323.149,A -85,B 0,C 180,E1 -11607.928,E2 -11607.928} C_VEL
LIN {X 0,Y 388.764,Z 323.566,A -85,B 0,C 180,E1 -11608.964,E2 -11608.964} C_VEL
LIN {X 0,Y 388.754,Z 323.595,A -85,B 0,C 180,E1 -11610,E2 -11610} C_VEL
LIN {X 0,Y 388.765,Z 323.238,A -85,B 0,C 180,E1 -11611.036,E2 -11611.036} C_VEL
LIN {X 0,Y 388.796,Z 322.482,A -85,B 0,C 180,E1 -11612.072,E2 -11612.072} C_VEL
LIN {X 0,Y 388.727,Z 319.658,A -85,B 0,C 180,E1 -11614.147,E2 -11614.147} C_VEL
LIN {X 0,Y 388.699,Z 316.388,A -85,B 0,C 180,E1 -11615.712,E2 -11615.712} C_VEL
LIN {X 0,Y 388.853,Z 312.066,A -85,B 0,C 180,E1 -11617.268,E2 -11617.268} C_VEL
LIN {X 0,Y 389.121,Z 306.528,A -85,B 0,C 180,E1 -11618.831,E2 -11618.831} C_VEL
LIN {X 0,Y 389.479,Z 299.598,A -85,B 0,C 180,E1 -11620.395,E2 -11620.395} C_VEL
LIN {X 0,Y 390.165,Z 290.941,A -85,B 0,C 180,E1 -11621.955,E2 -11621.955} C_VEL
LIN {X 0,Y 390.86,Z 282.041,A -85,B 0,C 180,E1 -11623.253,E2 -11623.253} C_VEL
LIN {X 0,Y 391.618,Z 271.07,A -85,B 0,C 180,E1 -11624.551,E2 -11624.551} C_VEL
LIN {X 0,Y 392.447,Z 260.001,A -85,B 0,C 180,E1 -11625.582,E2 -11625.582} C_VEL
LIN {X 0,Y 393.307,Z 247.584,A -85,B 0,C 180,E1 -11626.479,E2 -11626.479} C_VEL
LIN {X 0,Y 393.941,Z 235.801,A -85,B 0,C 180,E1 -11627.119,E2 -11627.119} C_VEL
LIN {X 0,Y 394.579,Z 223.15,A -85,B 0,C 180,E1 -11627.592,E2 -11627.592} C_VEL
LIN {X 0,Y 394.897,Z 206.936,A -85,B 0,C 180,E1 -11627.945,E2 -11627.945} C_VEL
LIN {X 0,Y 395.602,Z 141.181,A -85,B 0,C 180,E1 -11629.135,E2 -11629.135} C_VEL
LIN {X 0,Y 391.413,Z 110.453,A -85,B 0,C 180,E1 -11629.908,E2 -11629.908} C_VEL
LIN {X 0,Y 392.68,Z 91.556,A -85,B 0,C 180,E1 -11633.708,E2 -11633.708} C_VEL
LIN {X 0,Y 393.113,Z 84.578,A -85,B 0,C 180,E1 -11635.125,E2 -11635.125} C_VEL
LIN {X 0,Y 390.794,Z 72.066,A -85,B 0,C 180,E1 -11637.877,E2 -11637.877} C_VEL
LIN {X 0,Y 390.151,Z 68.887,A -85,B 0,C 180,E1 -11638.625,E2 -11638.625} C_VEL
LIN {X 0,Y 390.043,Z 68.896,A -85,B 0,C 180,E1 -11642.721,E2 -11642.721} C_VEL
LIN {X 0,Y 390.057,Z 68.901,A -85,B 0,C 180,E1 -11645.825,E2 -11645.825} C_VEL
LIN {X 0,Y 390.072,Z 68.894,A -85,B 0,C 180,E1 -11649.219,E2 -11649.219} C_VEL
LIN {X 0,Y 390.042,Z 68.896,A -85,B 0,C 180,E1 -11652.374,E2 -11652.374} C_VEL
LIN {X 0,Y 390.043,Z 68.901,A -85,B 0,C 180,E1 -11655.354,E2 -11655.354} C_VEL
LIN {X 0,Y 390.03,Z 68.898,A -85,B 0,C 180,E1 -11658.187,E2 -11658.187} C_VEL
LIN {X 0,Y 390.088,Z 68.893,A -85,B 0,C 180,E1 -11660.907,E2 -11660.907} C_VEL
LIN {X 0,Y 390.084,Z 68.893,A -85,B 0,C 180,E1 -11664.793,E2 -11664.793} C_VEL
LIN {X 0,Y 390.023,Z 68.9,A -85,B 0,C 180,E1 -11668.496,E2 -11668.496} C_VEL
LIN {X 0,Y 390.116,Z 68.887,A -85,B 0,C 180,E1 -11672.07,E2 -11672.07} C_VEL
LIN {X 0,Y 390.079,Z 68.892,A -85,B 0,C 180,E1 -11675.519,E2 -11675.519} C_VEL
LIN {X 0,Y 390.055,Z 68.9,A -85,B 0,C 180,E1 -11678.878,E2 -11678.878} C_VEL
LIN {X 0,Y 390.125,Z 68.887,A -85,B 0,C 180,E1 -11682.167,E2 -11682.167} C_VEL
LIN {X 0,Y 390.143,Z 68.884,A -85,B 0,C 180,E1 -11685.393,E2 -11685.393} C_VEL
LIN {X 0,Y 390.147,Z 68.888,A -85,B 0,C 180,E1 -11688.571,E2 -11688.571} C_VEL
LIN {X 0,Y 390.307,Z 68.866,A -85,B 0,C 180,E1 -11692.032,E2 -11692.032} C_VEL
LIN {X 0,Y 390.223,Z 68.875,A -85,B 0,C 180,E1 -11694.834,E2 -11694.834} C_VEL
LIN {X 0,Y 390.415,Z 68.854,A -85,B 0,C 180,E1 -11697.937,E2 -11697.937} C_VEL
LIN {X 0,Y 390.546,Z 68.839,A -85,B 0,C 180,E1 -11700,E2 -11700} C_VEL
LIN {X 0,Y 390.303,Z 68.864,A -85,B 0,C 180,E1 -11703.097,E2 -11703.097} C_VEL
LIN {X 0,Y 390.283,Z 68.867,A -85,B 0,C 180,E1 -11706.492,E2 -11706.492} C_VEL
LIN {X 0,Y 390.193,Z 68.879,A -85,B 0,C 180,E1 -11709.329,E2 -11709.329} C_VEL
LIN {X 0,Y 390.171,Z 68.88,A -85,B 0,C 180,E1 -11712.483,E2 -11712.483} C_VEL
LIN {X 0,Y 390.139,Z 68.89,A -85,B 0,C 180,E1 -11715.677,E2 -11715.677} C_VEL
LIN {X 0,Y 390.104,Z 68.89,A -85,B 0,C 180,E1 -11718.922,E2 -11718.922} C_VEL
LIN {X 0,Y 390.047,Z 68.896,A -85,B 0,C 180,E1 -11722.234,E2 -11722.234} C_VEL
LIN {X 0,Y 390.118,Z 68.889,A -85,B 0,C 180,E1 -11725.743,E2 -11725.743} C_VEL
LIN {X 0,Y 390.059,Z 68.9,A -85,B 0,C 180,E1 -11729.11,E2 -11729.11} C_VEL
LIN {X 0,Y 390.043,Z 68.899,A -85,B 0,C 180,E1 -11732.722,E2 -11732.722} C_VEL
LIN {X 0,Y 390.056,Z 68.894,A -85,B 0,C 180,E1 -11735.826,E2 -11735.826} C_VEL
LIN {X 0,Y 390.039,Z 68.899,A -85,B 0,C 180,E1 -11739.213,E2 -11739.213} C_VEL
LIN {X 0,Y 390.033,Z 68.9,A -85,B 0,C 180,E1 -11742.373,E2 -11742.373} C_VEL
LIN {X 0,Y 390.045,Z 68.896,A -85,B 0,C 180,E1 -11745.355,E2 -11745.355} C_VEL
LIN {X 0,Y 390.026,Z 68.901,A -85,B 0,C 180,E1 -11748.186,E2 -11748.186} C_VEL
LIN {X 0,Y 390.064,Z 68.896,A -85,B 0,C 180,E1 -11750.905,E2 -11750.905} C_VEL
LIN {X 0,Y 390.087,Z 68.893,A -85,B 0,C 180,E1 -11754.794,E2 -11754.794} C_VEL
LIN {X 0,Y 390.026,Z 68.902,A -85,B 0,C 180,E1 -11758.496,E2 -11758.496} C_VEL
LIN {X 0,Y 390.041,Z 68.902,A -85,B 0,C 180,E1 -11762.064,E2 -11762.064} C_VEL
LIN {X 0,Y 390.047,Z 68.897,A -85,B 0,C 180,E1 -11765.517,E2 -11765.517} C_VEL
LIN {X 0,Y 390.059,Z 68.894,A -85,B 0,C 180,E1 -11768.878,E2 -11768.878} C_VEL
LIN {X 0,Y 390.131,Z 68.892,A -85,B 0,C 180,E1 -11772.167,E2 -11772.167} C_VEL
LIN {X 0,Y 390.161,Z 69.032,A -85,B 0,C 180,E1 -11774.86,E2 -11774.86} C_VEL
LIN {X 0,Y 391.776,Z 78.093,A -85,B 0,C 180,E1 -11777.208,E2 -11777.208} C_VEL
LIN {X 0,Y 393.936,Z 87.227,A -85,B 0,C 180,E1 -11777.48,E2 -11777.48} C_VEL
LIN {X 0,Y 396.164,Z 99.27,A -85,B 0,C 180,E1 -11777.806,E2 -11777.806} C_VEL
LIN {X 0,Y 394.92,Z 184.649,A -85,B 0,C 180,E1 -11779.361,E2 -11779.361} C_VEL
LIN {X 0,Y 394.631,Z 197.861,A -85,B 0,C 180,E1 -11779.807,E2 -11779.807} C_VEL
LIN {X 0,Y 394.102,Z 210.538,A -85,B 0,C 180,E1 -11780.441,E2 -11780.441} C_VEL
LIN {X 0,Y 393.593,Z 222.588,A -85,B 0,C 180,E1 -11781.27,E2 -11781.27} C_VEL
LIN {X 0,Y 392.784,Z 234.048,A -85,B 0,C 180,E1 -11782.288,E2 -11782.288} C_VEL
LIN {X 0,Y 392.004,Z 244.363,A -85,B 0,C 180,E1 -11783.437,E2 -11783.437} C_VEL
LIN {X 0,Y 391.308,Z 252.806,A -85,B 0,C 180,E1 -11784.59,E2 -11784.59} C_VEL
LIN {X 0,Y 390.642,Z 260.598,A -85,B 0,C 180,E1 -11785.874,E2 -11785.874} C_VEL
LIN {X 0,Y 390.015,Z 268.214,A -85,B 0,C 180,E1 -11787.418,E2 -11787.418} C_VEL
LIN {X 0,Y 389.501,Z 274.336,A -85,B 0,C 180,E1 -11788.966,E2 -11788.966} C_VEL
LIN {X 0,Y 389.157,Z 279.202,A -85,B 0,C 180,E1 -11790.518,E2 -11790.518} C_VEL
LIN {X 0,Y 389.011,Z 282.956,A -85,B 0,C 180,E1 -11792.071,E2 -11792.071} C_VEL
LIN {X 0,Y 388.898,Z 284.899,A -85,B 0,C 180,E1 -11793.108,E2 -11793.108} C_VEL
LIN {X 0,Y 388.794,Z 286.435,A -85,B 0,C 180,E1 -11794.147,E2 -11794.147} C_VEL
LIN {X 0,Y 388.817,Z 287.521,A -85,B 0,C 180,E1 -11795.186,E2 -11795.186} C_VEL
LIN {X 0,Y 388.797,Z 288.446,A -85,B 0,C 180,E1 -11797.014,E2 -11797.014} C_VEL
LIN {X 0,Y 388.085,Z 288.577,A -85,B 0,C 180,E1 -11797.878,E2 -11797.878} C_VEL
LIN {X 0,Y 385.197,Z 288.202,A -85,B 0,C 180,E1 -11799.281,E2 -11799.281} C_VEL
LIN {X 0,Y 382.85,Z 287.409,A -85,B 0,C 180,E1 -11800.411,E2 -11800.411} C_VEL
LIN {X 0,Y 381.947,Z 286.473,A -85,B 0,C 180,E1 -11801.279,E2 -11801.279} C_VEL
LIN {X 0,Y 381.928,Z 286.072,A -85,B 0,C 180,E1 -11801.571,E2 -11801.571} C_VEL
LIN {X 0,Y 382.253,Z 283.709,A -85,B 0,C 180,E1 -11802.979,E2 -11802.979} C_VEL
LIN {X 0,Y 382.702,Z 279.224,A -85,B 0,C 180,E1 -11804.898,E2 -11804.898} C_VEL
LIN {X 0,Y 383.308,Z 274.179,A -85,B 0,C 180,E1 -11806.511,E2 -11806.511} C_VEL
LIN {X 0,Y 384.047,Z 267.789,A -85,B 0,C 180,E1 -11808.126,E2 -11808.126} C_VEL
LIN {X 0,Y 384.982,Z 259.745,A -85,B 0,C 180,E1 -11809.739,E2 -11809.739} C_VEL
LIN {X 0,Y 385.95,Z 251.505,A -85,B 0,C 180,E1 -11811.078,E2 -11811.078} C_VEL
LIN {X 0,Y 386.94,Z 241.393,A -85,B 0,C 180,E1 -11812.422,E2 -11812.422} C_VEL
LIN {X 0,Y 387.94,Z 231.311,A -85,B 0,C 180,E1 -11813.488,E2 -11813.488} C_VEL
LIN {X 0,Y 388.871,Z 220.288,A -85,B 0,C 180,E1 -11814.42,E2 -11814.42} C_VEL
LIN {X 0,Y 389.786,Z 208.062,A -85,B 0,C 180,E1 -11815.212,E2 -11815.212} C_VEL
LIN {X 0,Y 390.393,Z 195.371,A -85,B 0,C 180,E1 -11815.81,E2 -11815.81} C_VEL
LIN {X 0,Y 390.856,Z 181.836,A -85,B 0,C 180,E1 -11816.208,E2 -11816.208} C_VEL
LIN {X 0,Y 392.15,Z 101.258,A -85,B 0,C 180,E1 -11817.709,E2 -11817.709} C_VEL
LIN {X 0,Y 389.128,Z 89.391,A -85,B 0,C 180,E1 -11818.138,E2 -11818.138} C_VEL
LIN {X 0,Y 384.925,Z 78.787,A -85,B 0,C 180,E1 -11818.631,E2 -11818.631} C_VEL
LIN {X 0,Y 382.993,Z 69.779,A -85,B 0,C 180,E1 -11821.225,E2 -11821.225} C_VEL
LIN {X 0,Y 383.014,Z 69.773,A -85,B 0,C 180,E1 -11824.669,E2 -11824.669} C_VEL
LIN {X 0,Y 382.995,Z 69.774,A -85,B 0,C 180,E1 -11827.902,E2 -11827.902} C_VEL
LIN {X 0,Y 382.963,Z 69.782,A -85,B 0,C 180,E1 -11831.351,E2 -11831.351} C_VEL
LIN {X 0,Y 382.991,Z 69.765,A -85,B 0,C 180,E1 -11834.302,E2 -11834.302} C_VEL
LIN {X 0,Y 382.985,Z 69.779,A -85,B 0,C 180,E1 -11837.236,E2 -11837.236} C_VEL
LIN {X 0,Y 382.986,Z 69.776,A -85,B 0,C 180,E1 -11840.419,E2 -11840.419} C_VEL
LIN {X 0,Y 383.015,Z 69.771,A -85,B 0,C 180,E1 -11844.043,E2 -11844.043} C_VEL
LIN {X 0,Y 382.984,Z 69.775,A -85,B 0,C 180,E1 -11847.579,E2 -11847.579} C_VEL
LIN {X 0,Y 382.976,Z 69.778,A -85,B 0,C 180,E1 -11850.298,E2 -11850.298} C_VEL
LIN {X 0,Y 383.005,Z 69.773,A -85,B 0,C 180,E1 -11854.045,E2 -11854.045} C_VEL
LIN {X 0,Y 382.989,Z 69.771,A -85,B 0,C 180,E1 -11857.334,E2 -11857.334} C_VEL
LIN {X 0,Y 383.062,Z 69.77,A -85,B 0,C 180,E1 -11860.716,E2 -11860.716} C_VEL
LIN {X 0,Y 383.08,Z 69.762,A -85,B 0,C 180,E1 -11864.026,E2 -11864.026} C_VEL
LIN {X 0,Y 383.139,Z 69.749,A -85,B 0,C 180,E1 -11867.284,E2 -11867.284} C_VEL
LIN {X 0,Y 383.145,Z 69.761,A -85,B 0,C 180,E1 -11870.497,E2 -11870.497} C_VEL
LIN {X 0,Y 383.233,Z 69.737,A -85,B 0,C 180,E1 -11873.683,E2 -11873.683} C_VEL
LIN {X 0,Y 383.38,Z 69.73,A -85,B 0,C 180,E1 -11877.899,E2 -11877.899} C_VEL
LIN {X 0,Y 383.376,Z 69.73,A -85,B 0,C 180,E1 -11882.101,E2 -11882.101} C_VEL
LIN {X 0,Y 383.242,Z 69.738,A -85,B 0,C 180,E1 -11886.317,E2 -11886.317} C_VEL
LIN {X 0,Y 383.145,Z 69.759,A -85,B 0,C 180,E1 -11889.502,E2 -11889.502} C_VEL
LIN {X 0,Y 383.129,Z 69.757,A -85,B 0,C 180,E1 -11893.536,E2 -11893.536} C_VEL
LIN {X 0,Y 383.096,Z 69.756,A -85,B 0,C 180,E1 -11897.069,E2 -11897.069} C_VEL
LIN {X 0,Y 383.032,Z 69.77,A -85,B 0,C 180,E1 -11900.647,E2 -11900.647} C_VEL
LIN {X 0,Y 383.035,Z 69.772,A -85,B 0,C 180,E1 -11903.807,E2 -11903.807} C_VEL
LIN {X 0,Y 383.082,Z 69.761,A -85,B 0,C 180,E1 -11906.123,E2 -11906.123} C_VEL
LIN {X 0,Y 382.995,Z 69.775,A -85,B 0,C 180,E1 -11909.7,E2 -11909.7} C_VEL
LIN {X 0,Y 383.006,Z 69.775,A -85,B 0,C 180,E1 -11913.4,E2 -11913.4} C_VEL
LIN {X 0,Y 383.034,Z 69.753,A -85,B 0,C 180,E1 -11916.164,E2 -11916.164} C_VEL
LIN {X 0,Y 383.01,Z 69.774,A -85,B 0,C 180,E1 -11919.958,E2 -11919.958} C_VEL
LIN {X 0,Y 383.007,Z 69.778,A -85,B 0,C 180,E1 -11922.778,E2 -11922.778} C_VEL
LIN {X 0,Y 382.999,Z 69.774,A -85,B 0,C 180,E1 -11925.789,E2 -11925.789} C_VEL
LIN {X 0,Y 382.991,Z 69.776,A -85,B 0,C 180,E1 -11928.795,E2 -11928.795} C_VEL
LIN {X 0,Y 383.002,Z 69.775,A -85,B 0,C 180,E1 -11932.096,E2 -11932.096} C_VEL
LIN {X 0,Y 383.02,Z 69.773,A -85,B 0,C 180,E1 -11935.332,E2 -11935.332} C_VEL
LIN {X 0,Y 382.986,Z 69.784,A -85,B 0,C 180,E1 -11939.081,E2 -11939.081} C_VEL
LIN {X 0,Y 383.003,Z 69.889,A -85,B 0,C 180,E1 -11939.387,E2 -11939.387} C_VEL
LIN {X 0,Y 385.8,Z 81.722,A -85,B 0,C 180,E1 -11942.32,E2 -11942.32} C_VEL
LIN {X 0,Y 387.339,Z 89.61,A -85,B 0,C 180,E1 -11944.185,E2 -11944.185} C_VEL
LIN {X 0,Y 387.307,Z 92.499,A -85,B 0,C 180,E1 -11944.816,E2 -11944.816} C_VEL
LIN {X 0,Y 385.676,Z 109.829,A -85,B 0,C 180,E1 -11948.463,E2 -11948.463} C_VEL
LIN {X 0,Y 390.629,Z 137.064,A -85,B 0,C 180,E1 -11949.319,E2 -11949.319} C_VEL
LIN {X 0,Y 391.516,Z 145.121,A -85,B 0,C 180,E1 -11949.53,E2 -11949.53} C_VEL
LIN {X 0,Y 390.305,Z 218.944,A -85,B 0,C 180,E1 -11950.924,E2 -11950.924} C_VEL
LIN {X 0,Y 389.646,Z 231.877,A -85,B 0,C 180,E1 -11951.361,E2 -11951.361} C_VEL
LIN {X 0,Y 388.773,Z 243.982,A -85,B 0,C 180,E1 -11951.966,E2 -11951.966} C_VEL
LIN {X 0,Y 387.775,Z 255.407,A -85,B 0,C 180,E1 -11952.735,E2 -11952.735} C_VEL
LIN {X 0,Y 386.584,Z 267.151,A -85,B 0,C 180,E1 -11953.768,E2 -11953.768} C_VEL
LIN {X 0,Y 385.453,Z 277.695,A -85,B 0,C 180,E1 -11954.94,E2 -11954.94} C_VEL
LIN {X 0,Y 384.473,Z 287.22,A -85,B 0,C 180,E1 -11956.253,E2 -11956.253} C_VEL
LIN {X 0,Y 383.476,Z 296.41,A -85,B 0,C 180,E1 -11957.833,E2 -11957.833} C_VEL
LIN {X 0,Y 382.648,Z 303.822,A -85,B 0,C 180,E1 -11959.416,E2 -11959.416} C_VEL
LIN {X 0,Y 382.145,Z 309.792,A -85,B 0,C 180,E1 -11961.006,E2 -11961.006} C_VEL
LIN {X 0,Y 381.83,Z 314.524,A -85,B 0,C 180,E1 -11962.597,E2 -11962.597} C_VEL
LIN {X 0,Y 381.668,Z 317.587,A -85,B 0,C 180,E1 -11963.908,E2 -11963.908} C_VEL
LIN {X 0,Y 381.623,Z 320.781,A -85,B 0,C 180,E1 -11965.775,E2 -11965.775} C_VEL
LIN {X 0,Y 381.579,Z 322.024,A -85,B 0,C 180,E1 -11966.832,E2 -11966.832} C_VEL
LIN {X 0,Y 381.654,Z 322.848,A -85,B 0,C 180,E1 -11967.889,E2 -11967.889} C_VEL
LIN {X 0,Y 381.695,Z 323.253,A -85,B 0,C 180,E1 -11968.945,E2 -11968.945} C_VEL
LIN {X 0,Y 381.697,Z 322.898,A -85,B 0,C 180,E1 -11971.055,E2 -11971.055} C_VEL
LIN {X 0,Y 381.696,Z 322.117,A -85,B 0,C 180,E1 -11972.11,E2 -11972.11} C_VEL
LIN {X 0,Y 381.657,Z 319.265,A -85,B 0,C 180,E1 -11974.224,E2 -11974.224} C_VEL
LIN {X 0,Y 381.606,Z 315.523,A -85,B 0,C 180,E1 -11976.004,E2 -11976.004} C_VEL
LIN {X 0,Y 381.803,Z 311.612,A -85,B 0,C 180,E1 -11977.403,E2 -11977.403} C_VEL
LIN {X 0,Y 382.037,Z 306.036,A -85,B 0,C 180,E1 -11978.996,E2 -11978.996} C_VEL
LIN {X 0,Y 382.443,Z 299.068,A -85,B 0,C 180,E1 -11980.589,E2 -11980.589} C_VEL
LIN {X 0,Y 383.187,Z 290.345,A -85,B 0,C 180,E1 -11982.176,E2 -11982.176} C_VEL
LIN {X 0,Y 383.914,Z 281.389,A -85,B 0,C 180,E1 -11983.497,E2 -11983.497} C_VEL
LIN {X 0,Y 384.562,Z 272.106,A -85,B 0,C 180,E1 -11984.624,E2 -11984.624} C_VEL
LIN {X 0,Y 385.314,Z 262.187,A -85,B 0,C 180,E1 -11985.607,E2 -11985.607} C_VEL
LIN {X 0,Y 386.213,Z 250.589,A -85,B 0,C 180,E1 -11986.519,E2 -11986.519} C_VEL
LIN {X 0,Y 386.944,Z 238.526,A -85,B 0,C 180,E1 -11987.234,E2 -11987.234} C_VEL
LIN {X 0,Y 387.636,Z 225.47,A -85,B 0,C 180,E1 -11987.781,E2 -11987.781} C_VEL
LIN {X 0,Y 387.947,Z 213.125,A -85,B 0,C 180,E1 -11988.107,E2 -11988.107} C_VEL
LIN {X 0,Y 388.711,Z 141.42,A -85,B 0,C 180,E1 -11989.429,E2 -11989.429} C_VEL
LIN {X 0,Y 384.455,Z 110.181,A -85,B 0,C 180,E1 -11990.224,E2 -11990.224} C_VEL
LIN {X 0,Y 385.807,Z 91.593,A -85,B 0,C 180,E1 -11994.032,E2 -11994.032} C_VEL
LIN {X 0,Y 386.204,Z 86.748,A -85,B 0,C 180,E1 -11995.03,E2 -11995.03} C_VEL
LIN {X 0,Y 384.591,Z 77.037,A -85,B 0,C 180,E1 -11997.184,E2 -11997.184} C_VEL
LIN {X 0,Y 383.083,Z 69.769,A -85,B 0,C 180,E1 -11998.863,E2 -11998.863} C_VEL
LIN {X 0,Y 382.987,Z 69.776,A -85,B 0,C 180,E1 -12002.422,E2 -12002.422} C_VEL
LIN {X 0,Y 383.026,Z 69.775,A -85,B 0,C 180,E1 -12005.955,E2 -12005.955} C_VEL
LIN {X 0,Y 383.016,Z 69.777,A -85,B 0,C 180,E1 -12009.587,E2 -12009.587} C_VEL
LIN {X 0,Y 383.004,Z 69.773,A -85,B 0,C 180,E1 -12012.778,E2 -12012.778} C_VEL
LIN {X 0,Y 382.996,Z 69.777,A -85,B 0,C 180,E1 -12015.789,E2 -12015.789} C_VEL
LIN {X 0,Y 382.987,Z 69.776,A -85,B 0,C 180,E1 -12018.796,E2 -12018.796} C_VEL
LIN {X 0,Y 382.998,Z 69.774,A -85,B 0,C 180,E1 -12022.096,E2 -12022.096} C_VEL
LIN {X 0,Y 383.017,Z 69.776,A -85,B 0,C 180,E1 -12025.332,E2 -12025.332} C_VEL
LIN {X 0,Y 382.982,Z 69.782,A -85,B 0,C 180,E1 -12029.081,E2 -12029.081} C_VEL
LIN {X 0,Y 383.056,Z 69.77,A -85,B 0,C 180,E1 -12032.698,E2 -12032.698} C_VEL
LIN {X 0,Y 383.051,Z 69.772,A -85,B 0,C 180,E1 -12035.04,E2 -12035.04} C_VEL
LIN {X 0,Y 382.992,Z 69.778,A -85,B 0,C 180,E1 -12038.469,E2 -12038.469} C_VEL
LIN {X 0,Y 383.06,Z 69.766,A -85,B 0,C 180,E1 -12041.826,E2 -12041.826} C_VEL
LIN {X 0,Y 383.109,Z 69.761,A -85,B 0,C 180,E1 -12045.118,E2 -12045.118} C_VEL
LIN {X 0,Y 383.097,Z 69.767,A -85,B 0,C 180,E1 -12048.358,E2 -12048.358} C_VEL
LIN {X 0,Y 383.263,Z 69.743,A -85,B 0,C 180,E1 -12051.976,E2 -12051.976} C_VEL
LIN {X 0,Y 383.195,Z 69.751,A -85,B 0,C 180,E1 -12054.739,E2 -12054.739} C_VEL
LIN {X 0,Y 383.382,Z 69.729,A -85,B 0,C 180,E1 -12057.899,E2 -12057.899} C_VEL
LIN {X 0,Y 383.515,Z 69.715,A -85,B 0,C 180,E1 -12060,E2 -12060} C_VEL
LIN {X 0,Y 383.239,Z 69.744,A -85,B 0,C 180,E1 -12063.154,E2 -12063.154} C_VEL
LIN {X 0,Y 383.247,Z 69.744,A -85,B 0,C 180,E1 -12066.479,E2 -12066.479} C_VEL
LIN {X 0,Y 383.143,Z 69.759,A -85,B 0,C 180,E1 -12069.503,E2 -12069.503} C_VEL
LIN {X 0,Y 383.136,Z 69.756,A -85,B 0,C 180,E1 -12072.716,E2 -12072.716} C_VEL
LIN {X 0,Y 383.08,Z 69.766,A -85,B 0,C 180,E1 -12075.974,E2 -12075.974} C_VEL
LIN {X 0,Y 383.06,Z 69.77,A -85,B 0,C 180,E1 -12079.284,E2 -12079.284} C_VEL
LIN {X 0,Y 383.012,Z 69.772,A -85,B 0,C 180,E1 -12082.665,E2 -12082.665} C_VEL
LIN {X 0,Y 383.079,Z 69.764,A -85,B 0,C 180,E1 -12086.124,E2 -12086.124} C_VEL
LIN {X 0,Y 382.992,Z 69.776,A -85,B 0,C 180,E1 -12089.7,E2 -12089.7} C_VEL
LIN {X 0,Y 383.004,Z 69.776,A -85,B 0,C 180,E1 -12093.401,E2 -12093.401} C_VEL
LIN {X 0,Y 383.032,Z 69.77,A -85,B 0,C 180,E1 -12096.165,E2 -12096.165} C_VEL
LIN {X 0,Y 382.976,Z 69.776,A -85,B 0,C 180,E1 -12099.963,E2 -12099.963} C_VEL
LIN {X 0,Y 383.006,Z 69.779,A -85,B 0,C 180,E1 -12102.779,E2 -12102.779} C_VEL
LIN {X 0,Y 382.998,Z 69.774,A -85,B 0,C 180,E1 -12105.79,E2 -12105.79} C_VEL
LIN {X 0,Y 382.972,Z 69.781,A -85,B 0,C 180,E1 -12108.799,E2 -12108.799} C_VEL
LIN {X 0,Y 382.996,Z 69.777,A -85,B 0,C 180,E1 -12112.098,E2 -12112.098} C_VEL
LIN {X 0,Y 383.02,Z 69.771,A -85,B 0,C 180,E1 -12115.333,E2 -12115.333} C_VEL
LIN {X 0,Y 382.985,Z 69.775,A -85,B 0,C 180,E1 -12119.082,E2 -12119.082} C_VEL
LIN {X 0,Y 382.995,Z 69.775,A -85,B 0,C 180,E1 -12122.694,E2 -12122.694} C_VEL
LIN {X 0,Y 383.014,Z 69.776,A -85,B 0,C 180,E1 -12126.192,E2 -12126.192} C_VEL
LIN {X 0,Y 383.059,Z 69.769,A -85,B 0,C 180,E1 -12129.599,E2 -12129.599} C_VEL
LIN {X 0,Y 383.109,Z 69.763,A -85,B 0,C 180,E1 -12132.932,E2 -12132.932} C_VEL
LIN {X 0,Y 383.133,Z 69.93,A -85,B 0,C 180,E1 -12134.643,E2 -12134.643} C_VEL
LIN {X 0,Y 384.668,Z 78.328,A -85,B 0,C 180,E1 -12136.866,E2 -12136.866} C_VEL
LIN {X 0,Y 387.104,Z 87.787,A -85,B 0,C 180,E1 -12137.173,E2 -12137.173} C_VEL
LIN {X 0,Y 389.384,Z 100.052,A -85,B 0,C 180,E1 -12137.513,E2 -12137.513} C_VEL
LIN {X 0,Y 388.087,Z 185.642,A -85,B 0,C 180,E1 -12139.105,E2 -12139.105} C_VEL
LIN {X 0,Y 387.715,Z 199.393,A -85,B 0,C 180,E1 -12139.59,E2 -12139.59} C_VEL
LIN {X 0,Y 387.184,Z 212.254,A -85,B 0,C 180,E1 -12140.268,E2 -12140.268} C_VEL
LIN {X 0,Y 386.634,Z 223.927,A -85,B 0,C 180,E1 -12141.112,E2 -12141.112} C_VEL
LIN {X 0,Y 385.812,Z 235.199,A -85,B 0,C 180,E1 -12142.148,E2 -12142.148} C_VEL
LIN {X 0,Y 385.001,Z 245.368,A -85,B 0,C 180,E1 -12143.318,E2 -12143.318} C_VEL
LIN {X 0,Y 384.149,Z 255.314,A -85,B 0,C 180,E1 -12144.752,E2 -12144.752} C_VEL
LIN {X 0,Y 383.364,Z 264.066,A -85,B 0,C 180,E1 -12146.321,E2 -12146.321} C_VEL
LIN {X 0,Y 382.757,Z 271.091,A -85,B 0,C 180,E1 -12147.896,E2 -12147.896} C_VEL
LIN {X 0,Y 382.305,Z 276.696,A -85,B 0,C 180,E1 -12149.474,E2 -12149.474} C_VEL
LIN {X 0,Y 382.046,Z 281.114,A -85,B 0,C 180,E1 -12151.054,E2 -12151.054} C_VEL
LIN {X 0,Y 381.932,Z 283.449,A -85,B 0,C 180,E1 -12152.109,E2 -12152.109} C_VEL
LIN {X 0,Y 381.796,Z 285.366,A -85,B 0,C 180,E1 -12153.166,E2 -12153.166} C_VEL
LIN {X 0,Y 381.714,Z 286.861,A -85,B 0,C 180,E1 -12154.224,E2 -12154.224} C_VEL
LIN {X 0,Y 381.764,Z 288.513,A -85,B 0,C 180,E1 -12156.221,E2 -12156.221} C_VEL
LIN {X 0,Y 381.684,Z 288.856,A -85,B 0,C 180,E1 -12157.406,E2 -12157.406} C_VEL
LIN {X 0,Y 381.676,Z 288.747,A -85,B 0,C 180,E1 -12158.471,E2 -12158.471} C_VEL
LIN {X 0,Y 381.758,Z 287.271,A -85,B 0,C 180,E1 -12160.609,E2 -12160.609} C_VEL
LIN {X 0,Y 381.928,Z 286.072,A -85,B 0,C 180,E1 -12161.571,E2 -12161.571} C_VEL
LIN {X 0,Y 381.464,Z 284.87,A -85,B 0,C 180,E1 -12162.436,E2 -12162.436} C_VEL
LIN {X 0,Y 378.935,Z 282.379,A -85,B 0,C 180,E1 -12163.831,E2 -12163.831} C_VEL
LIN {X 0,Y 376.813,Z 279.859,A -85,B 0,C 180,E1 -12164.933,E2 -12164.933} C_VEL
LIN {X 0,Y 376.032,Z 277.617,A -85,B 0,C 180,E1 -12165.761,E2 -12165.761} C_VEL
LIN {X 0,Y 376.043,Z 276.774,A -85,B 0,C 180,E1 -12166.035,E2 -12166.035} C_VEL
LIN {X 0,Y 376.637,Z 272.182,A -85,B 0,C 180,E1 -12167.371,E2 -12167.371} C_VEL
LIN {X 0,Y 377.44,Z 265.223,A -85,B 0,C 180,E1 -12169.018,E2 -12169.018} C_VEL
LIN {X 0,Y 378.586,Z 256.44,A -85,B 0,C 180,E1 -12170.654,E2 -12170.654} C_VEL
LIN {X 0,Y 379.699,Z 246.756,A -85,B 0,C 180,E1 -12172.106,E2 -12172.106} C_VEL
LIN {X 0,Y 380.687,Z 237.396,A -85,B 0,C 180,E1 -12173.242,E2 -12173.242} C_VEL
LIN {X 0,Y 381.72,Z 226.222,A -85,B 0,C 180,E1 -12174.328,E2 -12174.328} C_VEL
LIN {X 0,Y 382.796,Z 213.639,A -85,B 0,C 180,E1 -12175.269,E2 -12175.269} C_VEL
LIN {X 0,Y 383.484,Z 202.484,A -85,B 0,C 180,E1 -12175.898,E2 -12175.898} C_VEL
LIN {X 0,Y 384.083,Z 189.818,A -85,B 0,C 180,E1 -12176.395,E2 -12176.395} C_VEL
LIN {X 0,Y 384.443,Z 172.291,A -85,B 0,C 180,E1 -12176.792,E2 -12176.792} C_VEL
LIN {X 0,Y 385.657,Z 102.567,A -85,B 0,C 180,E1 -12178.103,E2 -12178.103} C_VEL
LIN {X 0,Y 383.013,Z 92.156,A -85,B 0,C 180,E1 -12178.488,E2 -12178.488} C_VEL
LIN {X 0,Y 377.802,Z 79.063,A -85,B 0,C 180,E1 -12179.132,E2 -12179.132} C_VEL
LIN {X 0,Y 375.95,Z 70.658,A -85,B 0,C 180,E1 -12181.602,E2 -12181.602} C_VEL
LIN {X 0,Y 375.952,Z 70.655,A -85,B 0,C 180,E1 -12185.417,E2 -12185.417} C_VEL
LIN {X 0,Y 375.937,Z 70.656,A -85,B 0,C 180,E1 -12188.262,E2 -12188.262} C_VEL
LIN {X 0,Y 375.916,Z 70.659,A -85,B 0,C 180,E1 -12191.597,E2 -12191.597} C_VEL
LIN {X 0,Y 375.922,Z 70.644,A -85,B 0,C 180,E1 -12194.73,E2 -12194.73} C_VEL
LIN {X 0,Y 375.91,Z 70.66,A -85,B 0,C 180,E1 -12197.696,E2 -12197.696} C_VEL
LIN {X 0,Y 375.935,Z 70.655,A -85,B 0,C 180,E1 -12200.533,E2 -12200.533} C_VEL
LIN {X 0,Y 375.959,Z 70.655,A -85,B 0,C 180,E1 -12203.497,E2 -12203.497} C_VEL
LIN {X 0,Y 375.96,Z 70.654,A -85,B 0,C 180,E1 -12205.888,E2 -12205.888} C_VEL
LIN {X 0,Y 375.962,Z 70.654,A -85,B 0,C 180,E1 -12209.687,E2 -12209.687} C_VEL
LIN {X 0,Y 375.918,Z 70.652,A -85,B 0,C 180,E1 -12212.135,E2 -12212.135} C_VEL
LIN {X 0,Y 375.97,Z 70.649,A -85,B 0,C 180,E1 -12215.716,E2 -12215.716} C_VEL
LIN {X 0,Y 376.002,Z 70.65,A -85,B 0,C 180,E1 -12219.198,E2 -12219.198} C_VEL
LIN {X 0,Y 376.036,Z 70.636,A -85,B 0,C 180,E1 -12222.6,E2 -12222.6} C_VEL
LIN {X 0,Y 376.093,Z 70.638,A -85,B 0,C 180,E1 -12226.342,E2 -12226.342} C_VEL
LIN {X 0,Y 376.115,Z 70.634,A -85,B 0,C 180,E1 -12230.318,E2 -12230.318} C_VEL
LIN {X 0,Y 376.193,Z 70.614,A -85,B 0,C 180,E1 -12233.564,E2 -12233.564} C_VEL
LIN {X 0,Y 376.345,Z 70.606,A -85,B 0,C 180,E1 -12237.859,E2 -12237.859} C_VEL
LIN {X 0,Y 376.341,Z 70.607,A -85,B 0,C 180,E1 -12242.14,E2 -12242.14} C_VEL
LIN {X 0,Y 376.201,Z 70.615,A -85,B 0,C 180,E1 -12246.436,E2 -12246.436} C_VEL
LIN {X 0,Y 376.115,Z 70.635,A -85,B 0,C 180,E1 -12249.681,E2 -12249.681} C_VEL
LIN {X 0,Y 376.093,Z 70.635,A -85,B 0,C 180,E1 -12253.657,E2 -12253.657} C_VEL
LIN {X 0,Y 376.035,Z 70.636,A -85,B 0,C 180,E1 -12257.4,E2 -12257.4} C_VEL
LIN {X 0,Y 375.981,Z 70.649,A -85,B 0,C 180,E1 -12260.832,E2 -12260.832} C_VEL
LIN {X 0,Y 375.995,Z 70.647,A -85,B 0,C 180,E1 -12264.281,E2 -12264.281} C_VEL
LIN {X 0,Y 376.022,Z 70.641,A -85,B 0,C 180,E1 -12266.652,E2 -12266.652} C_VEL
LIN {X 0,Y 375.967,Z 70.649,A -85,B 0,C 180,E1 -12270.312,E2 -12270.312} C_VEL
LIN {X 0,Y 375.962,Z 70.65,A -85,B 0,C 180,E1 -12274.111,E2 -12274.111} C_VEL
LIN {X 0,Y 375.956,Z 70.634,A -85,B 0,C 180,E1 -12276.741,E2 -12276.741} C_VEL
LIN {X 0,Y 375.99,Z 70.649,A -85,B 0,C 180,E1 -12279.97,E2 -12279.97} C_VEL
LIN {X 0,Y 375.932,Z 70.656,A -85,B 0,C 180,E1 -12283.766,E2 -12283.766} C_VEL
LIN {X 0,Y 375.936,Z 70.656,A -85,B 0,C 180,E1 -12286.81,E2 -12286.81} C_VEL
LIN {X 0,Y 375.966,Z 70.65,A -85,B 0,C 180,E1 -12290.537,E2 -12290.537} C_VEL
LIN {X 0,Y 375.966,Z 70.652,A -85,B 0,C 180,E1 -12293.495,E2 -12293.495} C_VEL
LIN {X 0,Y 375.962,Z 70.656,A -85,B 0,C 180,E1 -12295.888,E2 -12295.888} C_VEL
LIN {X 0,Y 375.959,Z 70.731,A -85,B 0,C 180,E1 -12298.963,E2 -12298.963} C_VEL
LIN {X 0,Y 378.849,Z 82.968,A -85,B 0,C 180,E1 -12302.068,E2 -12302.068} C_VEL
LIN {X 0,Y 380.54,Z 92.163,A -85,B 0,C 180,E1 -12304.277,E2 -12304.277} C_VEL
LIN {X 0,Y 379.033,Z 107.879,A -85,B 0,C 180,E1 -12307.659,E2 -12307.659} C_VEL
LIN {X 0,Y 378.859,Z 109.491,A -85,B 0,C 180,E1 -12308.001,E2 -12308.001} C_VEL
LIN {X 0,Y 383.399,Z 133.905,A -85,B 0,C 180,E1 -12308.798,E2 -12308.798} C_VEL
LIN {X 0,Y 384.988,Z 145.488,A -85,B 0,C 180,E1 -12309.132,E2 -12309.132} C_VEL
LIN {X 0,Y 383.708,Z 219.008,A -85,B 0,C 180,E1 -12310.546,E2 -12310.546} C_VEL
LIN {X 0,Y 383.017,Z 231.862,A -85,B 0,C 180,E1 -12310.992,E2 -12310.992} C_VEL
LIN {X 0,Y 382.055,Z 244.449,A -85,B 0,C 180,E1 -12311.638,E2 -12311.638} C_VEL
LIN {X 0,Y 381.015,Z 255.661,A -85,B 0,C 180,E1 -12312.419,E2 -12312.419} C_VEL
LIN {X 0,Y 379.78,Z 267.278,A -85,B 0,C 180,E1 -12313.469,E2 -12313.469} C_VEL
LIN {X 0,Y 378.593,Z 277.743,A -85,B 0,C 180,E1 -12314.661,E2 -12314.661} C_VEL
LIN {X 0,Y 377.558,Z 287.195,A -85,B 0,C 180,E1 -12315.996,E2 -12315.996} C_VEL
LIN {X 0,Y 376.523,Z 296.32,A -85,B 0,C 180,E1 -12317.604,E2 -12317.604} C_VEL
LIN {X 0,Y 375.628,Z 303.69,A -85,B 0,C 180,E1 -12319.216,E2 -12319.216} C_VEL
LIN {X 0,Y 375.088,Z 309.624,A -85,B 0,C 180,E1 -12320.835,E2 -12320.835} C_VEL
LIN {X 0,Y 374.745,Z 314.322,A -85,B 0,C 180,E1 -12322.456,E2 -12322.456} C_VEL
LIN {X 0,Y 374.577,Z 317.651,A -85,B 0,C 180,E1 -12323.942,E2 -12323.942} C_VEL
LIN {X 0,Y 374.547,Z 320.52,A -85,B 0,C 180,E1 -12325.695,E2 -12325.695} C_VEL
LIN {X 0,Y 374.49,Z 321.749,A -85,B 0,C 180,E1 -12326.772,E2 -12326.772} C_VEL
LIN {X 0,Y 374.553,Z 322.546,A -85,B 0,C 180,E1 -12327.849,E2 -12327.849} C_VEL
LIN {X 0,Y 374.626,Z 322.939,A -85,B 0,C 180,E1 -12328.925,E2 -12328.925} C_VEL
LIN {X 0,Y 374.629,Z 322.559,A -85,B 0,C 180,E1 -12331.075,E2 -12331.075} C_VEL
LIN {X 0,Y 374.596,Z 321.749,A -85,B 0,C 180,E1 -12332.15,E2 -12332.15} C_VEL
LIN {X 0,Y 374.586,Z 318.87,A -85,B 0,C 180,E1 -12334.304,E2 -12334.304} C_VEL
LIN {X 0,Y 374.508,Z 315.467,A -85,B 0,C 180,E1 -12335.959,E2 -12335.959} C_VEL
LIN {X 0,Y 374.719,Z 311.152,A -85,B 0,C 180,E1 -12337.544,E2 -12337.544} C_VEL
LIN {X 0,Y 374.975,Z 305.541,A -85,B 0,C 180,E1 -12339.167,E2 -12339.167} C_VEL
LIN {X 0,Y 375.422,Z 298.531,A -85,B 0,C 180,E1 -12340.789,E2 -12340.789} C_VEL
LIN {X 0,Y 376.207,Z 289.743,A -85,B 0,C 180,E1 -12342.405,E2 -12342.405} C_VEL
LIN {X 0,Y 377.061,Z 279.745,A -85,B 0,C 180,E1 -12343.885,E2 -12343.885} C_VEL
LIN {X 0,Y 377.737,Z 269.566,A -85,B 0,C 180,E1 -12345.098,E2 -12345.098} C_VEL
LIN {X 0,Y 378.691,Z 258.27,A -85,B 0,C 180,E1 -12346.163,E2 -12346.163} C_VEL
LIN {X 0,Y 379.615,Z 245.568,A -85,B 0,C 180,E1 -12347.091,E2 -12347.091} C_VEL
LIN {X 0,Y 380.385,Z 233.175,A -85,B 0,C 180,E1 -12347.749,E2 -12347.749} C_VEL
LIN {X 0,Y 381.009,Z 219.372,A -85,B 0,C 180,E1 -12348.24,E2 -12348.24} C_VEL
LIN {X 0,Y 381.906,Z 142.144,A -85,B 0,C 180,E1 -12349.721,E2 -12349.721} C_VEL
LIN {X 0,Y 377.535,Z 109.734,A -85,B 0,C 180,E1 -12350.586,E2 -12350.586} C_VEL
LIN {X 0,Y 378.942,Z 91.497,A -85,B 0,C 180,E1 -12354.395,E2 -12354.395} C_VEL
LIN {X 0,Y 379.222,Z 87.534,A -85,B 0,C 180,E1 -12355.23,E2 -12355.23} C_VEL
LIN {X 0,Y 377.251,Z 76.419,A -85,B 0,C 180,E1 -12357.758,E2 -12357.758} C_VEL
LIN {X 0,Y 376.018,Z 70.649,A -85,B 0,C 180,E1 -12359.151,E2 -12359.151} C_VEL
LIN {X 0,Y 375.951,Z 70.651,A -85,B 0,C 180,E1 -12362.828,E2 -12362.828} C_VEL
LIN {X 0,Y 375.958,Z 70.653,A -85,B 0,C 180,E1 -12365.415,E2 -12365.415} C_VEL
LIN {X 0,Y 375.976,Z 70.65,A -85,B 0,C 180,E1 -12368.271,E2 -12368.271} C_VEL
LIN {X 0,Y 375.934,Z 70.66,A -85,B 0,C 180,E1 -12371.601,E2 -12371.601} C_VEL
LIN {X 0,Y 375.926,Z 70.658,A -85,B 0,C 180,E1 -12375.268,E2 -12375.268} C_VEL
LIN {X 0,Y 375.933,Z 70.654,A -85,B 0,C 180,E1 -12378.399,E2 -12378.399} C_VEL
LIN {X 0,Y 375.972,Z 70.651,A -85,B 0,C 180,E1 -12381.73,E2 -12381.73} C_VEL
LIN {X 0,Y 375.979,Z 70.653,A -85,B 0,C 180,E1 -12385.333,E2 -12385.333} C_VEL
LIN {X 0,Y 375.957,Z 70.651,A -85,B 0,C 180,E1 -12388.438,E2 -12388.438} C_VEL
LIN {X 0,Y 375.982,Z 70.648,A -85,B 0,C 180,E1 -12392.14,E2 -12392.14} C_VEL
LIN {X 0,Y 376.005,Z 70.647,A -85,B 0,C 180,E1 -12394.539,E2 -12394.539} C_VEL
LIN {X 0,Y 375.962,Z 70.65,A -85,B 0,C 180,E1 -12398.046,E2 -12398.046} C_VEL
LIN {X 0,Y 376.006,Z 70.645,A -85,B 0,C 180,E1 -12401.473,E2 -12401.473} C_VEL
LIN {X 0,Y 376.057,Z 70.642,A -85,B 0,C 180,E1 -12404.833,E2 -12404.833} C_VEL
LIN {X 0,Y 376.049,Z 70.642,A -85,B 0,C 180,E1 -12408.137,E2 -12408.137} C_VEL
LIN {X 0,Y 376.218,Z 70.62,A -85,B 0,C 180,E1 -12411.919,E2 -12411.919} C_VEL
LIN {X 0,Y 376.168,Z 70.627,A -85,B 0,C 180,E1 -12414.64,E2 -12414.64} C_VEL
LIN {X 0,Y 376.348,Z 70.605,A -85,B 0,C 180,E1 -12417.86,E2 -12417.86} C_VEL
LIN {X 0,Y 376.485,Z 70.59,A -85,B 0,C 180,E1 -12420,E2 -12420} C_VEL
LIN {X 0,Y 376.349,Z 70.607,A -85,B 0,C 180,E1 -12422.141,E2 -12422.141} C_VEL
LIN {X 0,Y 376.216,Z 70.62,A -85,B 0,C 180,E1 -12426.462,E2 -12426.462} C_VEL
LIN {X 0,Y 376.113,Z 70.637,A -85,B 0,C 180,E1 -12429.682,E2 -12429.682} C_VEL
LIN {X 0,Y 376.089,Z 70.641,A -85,B 0,C 180,E1 -12433.658,E2 -12433.658} C_VEL
LIN {X 0,Y 376.043,Z 70.646,A -85,B 0,C 180,E1 -12437.607,E2 -12437.607} C_VEL
LIN {X 0,Y 375.978,Z 70.649,A -85,B 0,C 180,E1 -12440.832,E2 -12440.832} C_VEL
LIN {X 0,Y 375.992,Z 70.646,A -85,B 0,C 180,E1 -12444.282,E2 -12444.282} C_VEL
LIN {X 0,Y 376.019,Z 70.644,A -85,B 0,C 180,E1 -12446.653,E2 -12446.653} C_VEL
LIN {X 0,Y 375.965,Z 70.65,A -85,B 0,C 180,E1 -12450.313,E2 -12450.313} C_VEL
LIN {X 0,Y 375.96,Z 70.65,A -85,B 0,C 180,E1 -12454.112,E2 -12454.112} C_VEL
LIN {X 0,Y 375.953,Z 70.656,A -85,B 0,C 180,E1 -12456.742,E2 -12456.742} C_VEL
LIN {X 0,Y 375.94,Z 70.653,A -85,B 0,C 180,E1 -12459.962,E2 -12459.962} C_VEL
LIN {X 0,Y 375.929,Z 70.654,A -85,B 0,C 180,E1 -12463.767,E2 -12463.767} C_VEL
LIN {X 0,Y 375.936,Z 70.658,A -85,B 0,C 180,E1 -12466.811,E2 -12466.811} C_VEL
LIN {X 0,Y 375.943,Z 70.659,A -85,B 0,C 180,E1 -12470.535,E2 -12470.535} C_VEL
LIN {X 0,Y 375.965,Z 70.65,A -85,B 0,C 180,E1 -12473.496,E2 -12473.496} C_VEL
LIN {X 0,Y 375.962,Z 70.652,A -85,B 0,C 180,E1 -12475.889,E2 -12475.889} C_VEL
LIN {X 0,Y 375.965,Z 70.651,A -85,B 0,C 180,E1 -12479.688,E2 -12479.688} C_VEL
LIN {X 0,Y 375.938,Z 70.66,A -85,B 0,C 180,E1 -12482.137,E2 -12482.137} C_VEL
LIN {X 0,Y 375.962,Z 70.653,A -85,B 0,C 180,E1 -12485.717,E2 -12485.717} C_VEL
LIN {X 0,Y 376.001,Z 70.646,A -85,B 0,C 180,E1 -12489.198,E2 -12489.198} C_VEL
LIN {X 0,Y 376.054,Z 70.645,A -85,B 0,C 180,E1 -12492.602,E2 -12492.602} C_VEL
LIN {X 0,Y 376.078,Z 70.825,A -85,B 0,C 180,E1 -12494.417,E2 -12494.417} C_VEL
LIN {X 0,Y 377.58,Z 78.619,A -85,B 0,C 180,E1 -12496.518,E2 -12496.518} C_VEL
LIN {X 0,Y 380.444,Z 89.192,A -85,B 0,C 180,E1 -12496.88,E2 -12496.88} C_VEL
LIN {X 0,Y 382.601,Z 100.599,A -85,B 0,C 180,E1 -12497.205,E2 -12497.205} C_VEL
LIN {X 0,Y 381.278,Z 185.483,A -85,B 0,C 180,E1 -12498.807,E2 -12498.807} C_VEL
LIN {X 0,Y 380.945,Z 198.63,A -85,B 0,C 180,E1 -12499.268,E2 -12499.268} C_VEL
LIN {X 0,Y 380.405,Z 210.716,A -85,B 0,C 180,E1 -12499.892,E2 -12499.892} C_VEL
LIN {X 0,Y 379.887,Z 222.087,A -85,B 0,C 180,E1 -12500.684,E2 -12500.684} C_VEL
LIN {X 0,Y 379.056,Z 233.783,A -85,B 0,C 180,E1 -12501.739,E2 -12501.739} C_VEL
LIN {X 0,Y 378.196,Z 244.257,A -85,B 0,C 180,E1 -12502.929,E2 -12502.929} C_VEL
LIN {X 0,Y 377.419,Z 252.827,A -85,B 0,C 180,E1 -12504.122,E2 -12504.122} C_VEL
LIN {X 0,Y 376.698,Z 260.722,A -85,B 0,C 180,E1 -12505.452,E2 -12505.452} C_VEL
LIN {X 0,Y 376.012,Z 268.466,A -85,B 0,C 180,E1 -12507.054,E2 -12507.054} C_VEL
LIN {X 0,Y 375.35,Z 275.561,A -85,B 0,C 180,E1 -12508.927,E2 -12508.927} C_VEL
LIN {X 0,Y 375.022,Z 280.301,A -85,B 0,C 180,E1 -12510.537,E2 -12510.537} C_VEL
LIN {X 0,Y 374.854,Z 283.94,A -85,B 0,C 180,E1 -12512.149,E2 -12512.149} C_VEL
LIN {X 0,Y 374.696,Z 285.831,A -85,B 0,C 180,E1 -12513.226,E2 -12513.226} C_VEL
LIN {X 0,Y 374.637,Z 287.273,A -85,B 0,C 180,E1 -12514.304,E2 -12514.304} C_VEL
LIN {X 0,Y 374.686,Z 288.815,A -85,B 0,C 180,E1 -12516.21,E2 -12516.21} C_VEL
LIN {X 0,Y 374.599,Z 289.191,A -85,B 0,C 180,E1 -12517.547,E2 -12517.547} C_VEL
LIN {X 0,Y 374.602,Z 289.031,A -85,B 0,C 180,E1 -12518.632,E2 -12518.632} C_VEL
LIN {X 0,Y 374.717,Z 287.502,A -85,B 0,C 180,E1 -12520.81,E2 -12520.81} C_VEL
LIN {X 0,Y 374.91,Z 286.143,A -85,B 0,C 180,E1 -12521.9,E2 -12521.9} C_VEL
LIN {X 0,Y 375.28,Z 283.256,A -85,B 0,C 180,E1 -12523.538,E2 -12523.538} C_VEL
LIN {X 0,Y 375.735,Z 279.314,A -85,B 0,C 180,E1 -12525.181,E2 -12525.181} C_VEL
LIN {X 0,Y 376.043,Z 276.774,A -85,B 0,C 180,E1 -12526.035,E2 -12526.035} C_VEL
LIN {X 0,Y 375.686,Z 274.233,A -85,B 0,C 180,E1 -12526.847,E2 -12526.847} C_VEL
LIN {X 0,Y 373.427,Z 269.788,A -85,B 0,C 180,E1 -12528.162,E2 -12528.162} C_VEL
LIN {X 0,Y 371.312,Z 264.727,A -85,B 0,C 180,E1 -12529.432,E2 -12529.432} C_VEL
LIN {X 0,Y 371.17,Z 261.199,A -85,B 0,C 180,E1 -12530.162,E2 -12530.162} C_VEL
LIN {X 0,Y 372.262,Z 252.794,A -85,B 0,C 180,E1 -12531.602,E2 -12531.602} C_VEL
LIN {X 0,Y 373.357,Z 242.511,A -85,B 0,C 180,E1 -12533.034,E2 -12533.034} C_VEL
LIN {X 0,Y 374.567,Z 231.552,A -85,B 0,C 180,E1 -12534.233,E2 -12534.233} C_VEL
LIN {X 0,Y 375.623,Z 220.438,A -85,B 0,C 180,E1 -12535.193,E2 -12535.193} C_VEL
LIN {X 0,Y 376.624,Z 207.816,A -85,B 0,C 180,E1 -12536.027,E2 -12536.027} C_VEL
LIN {X 0,Y 377.29,Z 195.116,A -85,B 0,C 180,E1 -12536.623,E2 -12536.623} C_VEL
LIN {X 0,Y 377.738,Z 182.267,A -85,B 0,C 180,E1 -12537.006,E2 -12537.006} C_VEL
LIN {X 0,Y 379.12,Z 103.483,A -85,B 0,C 180,E1 -12538.523,E2 -12538.523} C_VEL
LIN {X 0,Y 376.689,Z 94.23,A -85,B 0,C 180,E1 -12538.882,E2 -12538.882} C_VEL
LIN {X 0,Y 370.634,Z 79.353,A -85,B 0,C 180,E1 -12539.657,E2 -12539.657} C_VEL
LIN {X 0,Y 368.94,Z 71.529,A -85,B 0,C 180,E1 -12542.003,E2 -12542.003} C_VEL
LIN {X 0,Y 368.926,Z 71.528,A -85,B 0,C 180,E1 -12545,E2 -12545} C_VEL
LIN {X 0,Y 368.879,Z 71.537,A -85,B 0,C 180,E1 -12548.634,E2 -12548.634} C_VEL
LIN {X 0,Y 368.861,Z 71.539,A -85,B 0,C 180,E1 -12552.005,E2 -12552.005} C_VEL
LIN {X 0,Y 368.875,Z 71.522,A -85,B 0,C 180,E1 -12555.174,E2 -12555.174} C_VEL
LIN {X 0,Y 368.863,Z 71.534,A -85,B 0,C 180,E1 -12558.174,E2 -12558.174} C_VEL
LIN {X 0,Y 368.877,Z 71.534,A -85,B 0,C 180,E1 -12561.367,E2 -12561.367} C_VEL
LIN {X 0,Y 368.933,Z 71.525,A -85,B 0,C 180,E1 -12565.146,E2 -12565.146} C_VEL
LIN {X 0,Y 368.899,Z 71.528,A -85,B 0,C 180,E1 -12569.043,E2 -12569.043} C_VEL
LIN {X 0,Y 368.909,Z 71.528,A -85,B 0,C 180,E1 -12571.558,E2 -12571.558} C_VEL
LIN {X 0,Y 368.925,Z 71.531,A -85,B 0,C 180,E1 -12575.222,E2 -12575.222} C_VEL
LIN {X 0,Y 368.923,Z 71.53,A -85,B 0,C 180,E1 -12578.981,E2 -12578.981} C_VEL
LIN {X 0,Y 368.994,Z 71.513,A -85,B 0,C 180,E1 -12582.257,E2 -12582.257} C_VEL
LIN {X 0,Y 369.041,Z 71.515,A -85,B 0,C 180,E1 -12586.228,E2 -12586.228} C_VEL
LIN {X 0,Y 369.065,Z 71.51,A -85,B 0,C 180,E1 -12590.131,E2 -12590.131} C_VEL
LIN {X 0,Y 369.155,Z 71.49,A -85,B 0,C 180,E1 -12593.441,E2 -12593.441} C_VEL
LIN {X 0,Y 369.309,Z 71.482,A -85,B 0,C 180,E1 -12597.819,E2 -12597.819} C_VEL
LIN {X 0,Y 369.305,Z 71.484,A -85,B 0,C 180,E1 -12602.181,E2 -12602.181} C_VEL
LIN {X 0,Y 369.162,Z 71.493,A -85,B 0,C 180,E1 -12606.559,E2 -12606.559} C_VEL
LIN {X 0,Y 369.066,Z 71.51,A -85,B 0,C 180,E1 -12609.868,E2 -12609.868} C_VEL
LIN {X 0,Y 369.04,Z 71.515,A -85,B 0,C 180,E1 -12613.772,E2 -12613.772} C_VEL
LIN {X 0,Y 368.993,Z 71.514,A -85,B 0,C 180,E1 -12617.743,E2 -12617.743} C_VEL
LIN {X 0,Y 368.932,Z 71.526,A -85,B 0,C 180,E1 -12621.219,E2 -12621.219} C_VEL
LIN {X 0,Y 368.959,Z 71.525,A -85,B 0,C 180,E1 -12624.775,E2 -12624.775} C_VEL
LIN {X 0,Y 368.965,Z 71.52,A -85,B 0,C 180,E1 -12627.203,E2 -12627.203} C_VEL
LIN {X 0,Y 368.932,Z 71.525,A -85,B 0,C 180,E1 -12630.953,E2 -12630.953} C_VEL
LIN {X 0,Y 368.931,Z 71.517,A -85,B 0,C 180,E1 -12635.001,E2 -12635.001} C_VEL
LIN {X 0,Y 368.91,Z 71.527,A -85,B 0,C 180,E1 -12638.64,E2 -12638.64} C_VEL
LIN {X 0,Y 368.883,Z 71.533,A -85,B 0,C 180,E1 -12642.009,E2 -12642.009} C_VEL
LIN {X 0,Y 368.882,Z 71.533,A -85,B 0,C 180,E1 -12645.176,E2 -12645.176} C_VEL
LIN {X 0,Y 368.885,Z 71.532,A -85,B 0,C 180,E1 -12648.177,E2 -12648.177} C_VEL
LIN {X 0,Y 368.911,Z 71.529,A -85,B 0,C 180,E1 -12651.359,E2 -12651.359} C_VEL
LIN {X 0,Y 368.939,Z 71.524,A -85,B 0,C 180,E1 -12655.146,E2 -12655.146} C_VEL
LIN {X 0,Y 368.944,Z 71.602,A -85,B 0,C 180,E1 -12658.53,E2 -12658.53} C_VEL
LIN {X 0,Y 371.914,Z 84.214,A -85,B 0,C 180,E1 -12661.808,E2 -12661.808} C_VEL
LIN {X 0,Y 373.632,Z 93.401,A -85,B 0,C 180,E1 -12664.066,E2 -12664.066} C_VEL
LIN {X 0,Y 372.221,Z 107.791,A -85,B 0,C 180,E1 -12667.227,E2 -12667.227} C_VEL
LIN {X 0,Y 372.098,Z 109.15,A -85,B 0,C 180,E1 -12667.523,E2 -12667.523} C_VEL
LIN {X 0,Y 377.046,Z 135.819,A -85,B 0,C 180,E1 -12668.418,E2 -12668.418} C_VEL
LIN {X 0,Y 378.47,Z 145.881,A -85,B 0,C 180,E1 -12668.718,E2 -12668.718} C_VEL
LIN {X 0,Y 377.141,Z 217.921,A -85,B 0,C 180,E1 -12670.119,E2 -12670.119} C_VEL
LIN {X 0,Y 376.426,Z 231.105,A -85,B 0,C 180,E1 -12670.575,E2 -12670.575} C_VEL
LIN {X 0,Y 375.459,Z 243.8,A -85,B 0,C 180,E1 -12671.232,E2 -12671.232} C_VEL
LIN {X 0,Y 374.281,Z 255.899,A -85,B 0,C 180,E1 -12672.092,E2 -12672.092} C_VEL
LIN {X 0,Y 372.972,Z 267.411,A -85,B 0,C 180,E1 -12673.159,E2 -12673.159} C_VEL
LIN {X 0,Y 371.75,Z 277.797,A -85,B 0,C 180,E1 -12674.371,E2 -12674.371} C_VEL
LIN {X 0,Y 370.652,Z 287.166,A -85,B 0,C 180,E1 -12675.729,E2 -12675.729} C_VEL
LIN {X 0,Y 369.561,Z 296.234,A -85,B 0,C 180,E1 -12677.367,E2 -12677.367} C_VEL
LIN {X 0,Y 368.61,Z 303.562,A -85,B 0,C 180,E1 -12679.008,E2 -12679.008} C_VEL
LIN {X 0,Y 368.034,Z 309.457,A -85,B 0,C 180,E1 -12680.658,E2 -12680.658} C_VEL
LIN {X 0,Y 367.679,Z 314.122,A -85,B 0,C 180,E1 -12682.31,E2 -12682.31} C_VEL
LIN {X 0,Y 367.503,Z 317.668,A -85,B 0,C 180,E1 -12683.951,E2 -12683.951} C_VEL
LIN {X 0,Y 367.451,Z 320.26,A -85,B 0,C 180,E1 -12685.612,E2 -12685.612} C_VEL
LIN {X 0,Y 367.406,Z 321.472,A -85,B 0,C 180,E1 -12686.71,E2 -12686.71} C_VEL
LIN {X 0,Y 367.452,Z 322.245,A -85,B 0,C 180,E1 -12687.807,E2 -12687.807} C_VEL
LIN {X 0,Y 367.54,Z 322.626,A -85,B 0,C 180,E1 -12688.904,E2 -12688.904} C_VEL
LIN {X 0,Y 367.548,Z 322.616,A -85,B 0,C 180,E1 -12690,E2 -12690} C_VEL
LIN {X 0,Y 367.544,Z 322.217,A -85,B 0,C 180,E1 -12691.095,E2 -12691.095} C_VEL
LIN {X 0,Y 367.497,Z 321.38,A -85,B 0,C 180,E1 -12692.192,E2 -12692.192} C_VEL
LIN {X 0,Y 367.514,Z 318.473,A -85,B 0,C 180,E1 -12694.387,E2 -12694.387} C_VEL
LIN {X 0,Y 367.411,Z 315.407,A -85,B 0,C 180,E1 -12695.913,E2 -12695.913} C_VEL
LIN {X 0,Y 367.659,Z 310.692,A -85,B 0,C 180,E1 -12697.689,E2 -12697.689} C_VEL
LIN {X 0,Y 367.936,Z 305.045,A -85,B 0,C 180,E1 -12699.344,E2 -12699.344} C_VEL
LIN {X 0,Y 368.406,Z 297.983,A -85,B 0,C 180,E1 -12700.997,E2 -12700.997} C_VEL
LIN {X 0,Y 369.225,Z 289.136,A -85,B 0,C 180,E1 -12702.644,E2 -12702.644} C_VEL
LIN {X 0,Y 370.121,Z 279.079,A -85,B 0,C 180,E1 -12704.151,E2 -12704.151} C_VEL
LIN {X 0,Y 370.822,Z 268.787,A -85,B 0,C 180,E1 -12705.387,E2 -12705.387} C_VEL
LIN {X 0,Y 371.869,Z 257.393,A -85,B 0,C 180,E1 -12706.468,E2 -12706.468} C_VEL
LIN {X 0,Y 372.731,Z 245.547,A -85,B 0,C 180,E1 -12707.346,E2 -12707.346} C_VEL
LIN {X 0,Y 373.577,Z 232.544,A -85,B 0,C 180,E1 -12708.048,E2 -12708.048} C_VEL
LIN {X 0,Y 374.163,Z 219.724,A -85,B 0,C 180,E1 -12708.515,E2 -12708.515} C_VEL
LIN {X 0,Y 374.697,Z 187.747,A -85,B 0,C 180,E1 -12709.16,E2 -12709.16} C_VEL
LIN {X 0,Y 375.148,Z 143.098,A -85,B 0,C 180,E1 -12710.016,E2 -12710.016} C_VEL
LIN {X 0,Y 370.603,Z 109.473,A -85,B 0,C 180,E1 -12710.924,E2 -12710.924} C_VEL
LIN {X 0,Y 372.168,Z 90.41,A -85,B 0,C 180,E1 -12714.983,E2 -12714.983} C_VEL
LIN {X 0,Y 372.027,Z 86.935,A -85,B 0,C 180,E1 -12715.753,E2 -12715.753} C_VEL
LIN {X 0,Y 369.541,Z 74.214,A -85,B 0,C 180,E1 -12718.74,E2 -12718.74} C_VEL
LIN {X 0,Y 368.953,Z 71.528,A -85,B 0,C 180,E1 -12719.405,E2 -12719.405} C_VEL
LIN {X 0,Y 368.898,Z 71.53,A -85,B 0,C 180,E1 -12723.043,E2 -12723.043} C_VEL
LIN {X 0,Y 368.918,Z 71.53,A -85,B 0,C 180,E1 -12726.196,E2 -12726.196} C_VEL
LIN {X 0,Y 368.904,Z 71.53,A -85,B 0,C 180,E1 -12728.953,E2 -12728.953} C_VEL
LIN {X 0,Y 368.881,Z 71.534,A -85,B 0,C 180,E1 -12732.009,E2 -12732.009} C_VEL
LIN {X 0,Y 368.879,Z 71.535,A -85,B 0,C 180,E1 -12735.176,E2 -12735.176} C_VEL
LIN {X 0,Y 368.882,Z 71.532,A -85,B 0,C 180,E1 -12738.177,E2 -12738.177} C_VEL
LIN {X 0,Y 368.907,Z 71.535,A -85,B 0,C 180,E1 -12741.36,E2 -12741.36} C_VEL
LIN {X 0,Y 368.935,Z 71.531,A -85,B 0,C 180,E1 -12745.146,E2 -12745.146} C_VEL
LIN {X 0,Y 368.928,Z 71.533,A -85,B 0,C 180,E1 -12749.046,E2 -12749.046} C_VEL
LIN {X 0,Y 368.975,Z 71.522,A -85,B 0,C 180,E1 -12751.564,E2 -12751.564} C_VEL
LIN {X 0,Y 368.999,Z 71.517,A -85,B 0,C 180,E1 -12754.02,E2 -12754.02} C_VEL
LIN {X 0,Y 368.931,Z 71.526,A -85,B 0,C 180,E1 -12757.605,E2 -12757.605} C_VEL
LIN {X 0,Y 368.956,Z 71.525,A -85,B 0,C 180,E1 -12761.106,E2 -12761.106} C_VEL
LIN {X 0,Y 368.997,Z 71.524,A -85,B 0,C 180,E1 -12764.535,E2 -12764.535} C_VEL
LIN {X 0,Y 369.004,Z 71.518,A -85,B 0,C 180,E1 -12767.907,E2 -12767.907} C_VEL
LIN {X 0,Y 369.165,Z 71.499,A -85,B 0,C 180,E1 -12771.869,E2 -12771.869} C_VEL
LIN {X 0,Y 369.141,Z 71.503,A -85,B 0,C 180,E1 -12774.538,E2 -12774.538} C_VEL
LIN {X 0,Y 369.313,Z 71.481,A -85,B 0,C 180,E1 -12777.819,E2 -12777.819} C_VEL
LIN {X 0,Y 369.454,Z 71.466,A -85,B 0,C 180,E1 -12780,E2 -12780} C_VEL
LIN {X 0,Y 369.314,Z 71.483,A -85,B 0,C 180,E1 -12782.181,E2 -12782.181} C_VEL
LIN {X 0,Y 369.178,Z 71.496,A -85,B 0,C 180,E1 -12786.559,E2 -12786.559} C_VEL
LIN {X 0,Y 369.063,Z 71.515,A -85,B 0,C 180,E1 -12789.869,E2 -12789.869} C_VEL
LIN {X 0,Y 369.037,Z 71.518,A -85,B 0,C 180,E1 -12793.773,E2 -12793.773} C_VEL
LIN {X 0,Y 369.001,Z 71.521,A -85,B 0,C 180,E1 -12797.769,E2 -12797.769} C_VEL
LIN {X 0,Y 368.93,Z 71.53,A -85,B 0,C 180,E1 -12801.22,E2 -12801.22} C_VEL
LIN {X 0,Y 368.957,Z 71.524,A -85,B 0,C 180,E1 -12804.776,E2 -12804.776} C_VEL
LIN {X 0,Y 368.963,Z 71.528,A -85,B 0,C 180,E1 -12807.204,E2 -12807.204} C_VEL
LIN {X 0,Y 368.93,Z 71.531,A -85,B 0,C 180,E1 -12810.954,E2 -12810.954} C_VEL
LIN {X 0,Y 368.929,Z 71.532,A -85,B 0,C 180,E1 -12815.002,E2 -12815.002} C_VEL
LIN {X 0,Y 368.878,Z 71.536,A -85,B 0,C 180,E1 -12818.635,E2 -12818.635} C_VEL
LIN {X 0,Y 368.871,Z 71.534,A -85,B 0,C 180,E1 -12822.008,E2 -12822.008} C_VEL
LIN {X 0,Y 368.88,Z 71.534,A -85,B 0,C 180,E1 -12825.176,E2 -12825.176} C_VEL
LIN {X 0,Y 368.875,Z 71.535,A -85,B 0,C 180,E1 -12828.177,E2 -12828.177} C_VEL
LIN {X 0,Y 368.881,Z 71.532,A -85,B 0,C 180,E1 -12831.366,E2 -12831.366} C_VEL
LIN {X 0,Y 368.938,Z 71.525,A -85,B 0,C 180,E1 -12835.147,E2 -12835.147} C_VEL
LIN {X 0,Y 368.932,Z 71.526,A -85,B 0,C 180,E1 -12839.047,E2 -12839.047} C_VEL
LIN {X 0,Y 368.875,Z 71.534,A -85,B 0,C 180,E1 -12842.79,E2 -12842.79} C_VEL
LIN {X 0,Y 368.95,Z 71.526,A -85,B 0,C 180,E1 -12846.421,E2 -12846.421} C_VEL
LIN {X 0,Y 368.94,Z 71.53,A -85,B 0,C 180,E1 -12849.948,E2 -12849.948} C_VEL
LIN {X 0,Y 368.98,Z 71.523,A -85,B 0,C 180,E1 -12853.399,E2 -12853.399} C_VEL
LIN {X 0,Y 369.052,Z 71.742,A -85,B 0,C 180,E1 -12854.184,E2 -12854.184} C_VEL
LIN {X 0,Y 370.479,Z 79.152,A -85,B 0,C 180,E1 -12856.179,E2 -12856.179} C_VEL
LIN {X 0,Y 373.71,Z 90.139,A -85,B 0,C 180,E1 -12856.564,E2 -12856.564} C_VEL
LIN {X 0,Y 375.861,Z 102.221,A -85,B 0,C 180,E1 -12856.91,E2 -12856.91} C_VEL
LIN {X 0,Y 374.462,Z 186.425,A -85,B 0,C 180,E1 -12858.532,E2 -12858.532} C_VEL
LIN {X 0,Y 374.104,Z 199.37,A -85,B 0,C 180,E1 -12859.001,E2 -12859.001} C_VEL
LIN {X 0,Y 373.546,Z 211.346,A -85,B 0,C 180,E1 -12859.636,E2 -12859.636} C_VEL
LIN {X 0,Y 372.95,Z 223.445,A -85,B 0,C 180,E1 -12860.51,E2 -12860.51} C_VEL
LIN {X 0,Y 372.092,Z 234.919,A -85,B 0,C 180,E1 -12861.583,E2 -12861.583} C_VEL
LIN {X 0,Y 371.204,Z 245.253,A -85,B 0,C 180,E1 -12862.795,E2 -12862.795} C_VEL
LIN {X 0,Y 370.404,Z 253.711,A -85,B 0,C 180,E1 -12864.01,E2 -12864.01} C_VEL
LIN {X 0,Y 369.663,Z 261.513,A -85,B 0,C 180,E1 -12865.366,E2 -12865.366} C_VEL
LIN {X 0,Y 368.961,Z 269.14,A -85,B 0,C 180,E1 -12866.998,E2 -12866.998} C_VEL
LIN {X 0,Y 368.279,Z 276.169,A -85,B 0,C 180,E1 -12868.907,E2 -12868.907} C_VEL
LIN {X 0,Y 367.956,Z 280.847,A -85,B 0,C 180,E1 -12870.548,E2 -12870.548} C_VEL
LIN {X 0,Y 367.777,Z 284.431,A -85,B 0,C 180,E1 -12872.191,E2 -12872.191} C_VEL
LIN {X 0,Y 367.597,Z 286.291,A -85,B 0,C 180,E1 -12873.288,E2 -12873.288} C_VEL
LIN {X 0,Y 367.562,Z 287.683,A -85,B 0,C 180,E1 -12874.387,E2 -12874.387} C_VEL
LIN {X 0,Y 367.603,Z 289.112,A -85,B 0,C 180,E1 -12876.19,E2 -12876.19} C_VEL
LIN {X 0,Y 367.513,Z 289.52,A -85,B 0,C 180,E1 -12877.693,E2 -12877.693} C_VEL
LIN {X 0,Y 367.512,Z 289.315,A -85,B 0,C 180,E1 -12878.8,E2 -12878.8} C_VEL
LIN {X 0,Y 367.684,Z 287.733,A -85,B 0,C 180,E1 -12881.02,E2 -12881.02} C_VEL
LIN {X 0,Y 367.873,Z 286.336,A -85,B 0,C 180,E1 -12882.131,E2 -12882.131} C_VEL
LIN {X 0,Y 368.263,Z 283.4,A -85,B 0,C 180,E1 -12883.801,E2 -12883.801} C_VEL
LIN {X 0,Y 368.767,Z 279.399,A -85,B 0,C 180,E1 -12885.475,E2 -12885.475} C_VEL
LIN {X 0,Y 369.605,Z 273.192,A -85,B 0,C 180,E1 -12887.427,E2 -12887.427} C_VEL
LIN {X 0,Y 370.441,Z 266.393,A -85,B 0,C 180,E1 -12889.103,E2 -12889.103} C_VEL
LIN {X 0,Y 371.17,Z 261.199,A -85,B 0,C 180,E1 -12890.162,E2 -12890.162} C_VEL
LIN {X 0,Y 371.043,Z 257.488,A -85,B 0,C 180,E1 -12890.872,E2 -12890.872} C_VEL
LIN {X 0,Y 369.048,Z 251.268,A -85,B 0,C 180,E1 -12892.033,E2 -12892.033} C_VEL
LIN {X 0,Y 367.098,Z 244.556,A -85,B 0,C 180,E1 -12893.126,E2 -12893.126} C_VEL
LIN {X 0,Y 367.025,Z 240.037,A -85,B 0,C 180,E1 -12893.719,E2 -12893.719} C_VEL
LIN {X 0,Y 368.127,Z 229.514,A -85,B 0,C 180,E1 -12894.835,E2 -12894.835} C_VEL
LIN {X 0,Y 369.319,Z 217.787,A -85,B 0,C 180,E1 -12895.805,E2 -12895.805} C_VEL
LIN {X 0,Y 370.2,Z 205.484,A -85,B 0,C 180,E1 -12896.572,E2 -12896.572} C_VEL
LIN {X 0,Y 370.881,Z 192.911,A -85,B 0,C 180,E1 -12897.128,E2 -12897.128} C_VEL
LIN {X 0,Y 371.272,Z 180.169,A -85,B 0,C 180,E1 -12897.478,E2 -12897.478} C_VEL
LIN {X 0,Y 372.669,Z 104.777,A -85,B 0,C 180,E1 -12898.947,E2 -12898.947} C_VEL
LIN {X 0,Y 370.465,Z 96.561,A -85,B 0,C 180,E1 -12899.277,E2 -12899.277} C_VEL
LIN {X 0,Y 363.522,Z 79.73,A -85,B 0,C 180,E1 -12900.177,E2 -12900.177} C_VEL
LIN {X 0,Y 361.866,Z 72.409,A -85,B 0,C 180,E1 -12902.448,E2 -12902.448} C_VEL
LIN {X 0,Y 361.867,Z 72.411,A -85,B 0,C 180,E1 -12905.637,E2 -12905.637} C_VEL
LIN {X 0,Y 361.828,Z 72.415,A -85,B 0,C 180,E1 -12909.018,E2 -12909.018} C_VEL
LIN {X 0,Y 361.832,Z 72.413,A -85,B 0,C 180,E1 -12912.83,E2 -12912.83} C_VEL
LIN {X 0,Y 361.816,Z 72.409,A -85,B 0,C 180,E1 -12915.948,E2 -12915.948} C_VEL
LIN {X 0,Y 361.813,Z 72.413,A -85,B 0,C 180,E1 -12919.249,E2 -12919.249} C_VEL
LIN {X 0,Y 361.863,Z 72.409,A -85,B 0,C 180,E1 -12922.981,E2 -12922.981} C_VEL
LIN {X 0,Y 361.86,Z 72.409,A -85,B 0,C 180,E1 -12926.631,E2 -12926.631} C_VEL
LIN {X 0,Y 361.85,Z 72.412,A -85,B 0,C 180,E1 -12929.669,E2 -12929.669} C_VEL
LIN {X 0,Y 361.857,Z 72.408,A -85,B 0,C 180,E1 -12933.467,E2 -12933.467} C_VEL
LIN {X 0,Y 361.873,Z 72.405,A -85,B 0,C 180,E1 -12935.93,E2 -12935.93} C_VEL
LIN {X 0,Y 361.89,Z 72.405,A -85,B 0,C 180,E1 -12939.539,E2 -12939.539} C_VEL
LIN {X 0,Y 361.93,Z 72.395,A -85,B 0,C 180,E1 -12943.066,E2 -12943.066} C_VEL
LIN {X 0,Y 362.003,Z 72.389,A -85,B 0,C 180,E1 -12946.528,E2 -12946.528} C_VEL
LIN {X 0,Y 362.002,Z 72.389,A -85,B 0,C 180,E1 -12949.937,E2 -12949.937} C_VEL
LIN {X 0,Y 362.119,Z 72.366,A -85,B 0,C 180,E1 -12953.313,E2 -12953.313} C_VEL
LIN {X 0,Y 362.272,Z 72.358,A -85,B 0,C 180,E1 -12957.776,E2 -12957.776} C_VEL
LIN {X 0,Y 362.267,Z 72.361,A -85,B 0,C 180,E1 -12962.223,E2 -12962.223} C_VEL
LIN {X 0,Y 362.125,Z 72.369,A -85,B 0,C 180,E1 -12966.687,E2 -12966.687} C_VEL
LIN {X 0,Y 362.002,Z 72.388,A -85,B 0,C 180,E1 -12970.063,E2 -12970.063} C_VEL
LIN {X 0,Y 362.001,Z 72.393,A -85,B 0,C 180,E1 -12973.899,E2 -12973.899} C_VEL
LIN {X 0,Y 361.93,Z 72.392,A -85,B 0,C 180,E1 -12976.934,E2 -12976.934} C_VEL
LIN {X 0,Y 361.896,Z 72.402,A -85,B 0,C 180,E1 -12980.46,E2 -12980.46} C_VEL
LIN {X 0,Y 361.897,Z 72.404,A -85,B 0,C 180,E1 -12984.113,E2 -12984.113} C_VEL
LIN {X 0,Y 361.944,Z 72.394,A -85,B 0,C 180,E1 -12986.721,E2 -12986.721} C_VEL
LIN {X 0,Y 361.875,Z 72.405,A -85,B 0,C 180,E1 -12990.328,E2 -12990.328} C_VEL
LIN {X 0,Y 361.857,Z 72.408,A -85,B 0,C 180,E1 -12994.28,E2 -12994.28} C_VEL
LIN {X 0,Y 361.866,Z 72.391,A -85,B 0,C 180,E1 -12997.223,E2 -12997.223} C_VEL
LIN {X 0,Y 361.838,Z 72.411,A -85,B 0,C 180,E1 -13000.755,E2 -13000.755} C_VEL
LIN {X 0,Y 361.819,Z 72.416,A -85,B 0,C 180,E1 -13004.368,E2 -13004.368} C_VEL
LIN {X 0,Y 361.838,Z 72.41,A -85,B 0,C 180,E1 -13007.568,E2 -13007.568} C_VEL
LIN {X 0,Y 361.873,Z 72.407,A -85,B 0,C 180,E1 -13010.973,E2 -13010.973} C_VEL
